(* CoDeSys 2.3 library: TcMc2Drive.lib *)
(* Libraries: STANDARD.LIB 5.6.98 11:03:02, TcBase.lib 14.5.09 11:14:08, TcSystem.lib 10.9.09 11:54:20, TcUtilities.lib 13.10.09 07:46:56, TcEtherCAT.lib 15.1.10 19:43:55, TcTestAndSet.lib 23.2.09 11:50:08, TcDrive.lib 19.1.10 09:32:20, TcBaseMath.lib 27.7.04 11:07:56, TcMath.lib 23.9.04 14:15:30, TcMC2.lib 18.11.09 13:36:54 *)

(* POU F_GetVersionTcMc2Drive, ST *)
FUNCTION F_GetVersionTcMc2Drive : UINT
(* Returns the library version information  *)
VAR_INPUT
	nVersionElement       :       INT;
END_VAR
VAR
END_VAR
(* Version history:
Date          		| Version 		| created under 	     	| Author    | Remark 
------------------------------------------------------------------------------------------------------------------------------------------------------ 
15.05.2008    		| 0.0.1      	| V2.10.0 (Build 1325) 		| I.Ch.		| first release 
13.06.2008    		| 0.0.2      	| V2.10.0 (Build 1325) 		| I.Ch.		| FB_SoEAX5000Reset added  
10.07.2008    		| 0.0.3      	| V2.10.0 (Build 1326) 		| PKa		| FB_SoEAX5000Reset interface update/bugfix  
11.07.2008    		| 0.0.4      	| V2.10.0 (Build 1328) 		| PKa		| FB_SoEAX5000Reset AdsWrite call with falling edge, NC reset timer set to 1sec 
28.07.2008    		| 0.0.5      	| V2.10.0 (Build 1328) 		| I.Ch.		| using ST_DriveRef instead of ST_SoE_DriveRef
18.08.2008    		| 0.0.6      	| V2.10.0 (Build 1328) 		| I.Ch.		| Axis as VAR_IN_OUT
29.08.2008    		| 0.0.7      	| V2.10.0 (Build 1328) 		| I.Ch.		| FB_SoEAX5000Reset removed, FB_SoEReset modified
24.09.2008			| 0.0.8			| V2.10.0 (Build 1328)		| AnK		| FB_SoEReset: internal NC reset removed
02.10.2008			| 0.0.9			| V2.10.0 (Build 1328)		| I.Ch.		| folders added
03.10.2008			| 0.0.10		| V2.10.0 (Build 1330)		| I.Ch.		| created from TcNcDrive.lib v0.0.9
12.12.2008			| 0.0.11		| V2.10.0 (Build 1330)		| I.Ch.		| FB_SoEAX5000FirmwareUpdate added
15.12.2008			| 0.0.13		| V2.10.0 (Build 1330)		| I.Ch.		| cleanup
16.12.2008			| 0.0.14		| V2.10.0 (Build 1330)		| I.Ch.		| provide FB_EcFoeLoad.sInfo as iDiagNumber
16.01.2009			| 0.0.15		| V2.10.0 (Build 1331)		| I.Ch.		| update library list
05.02.2009			| 0.0.19		| V2.10.0 (Build 1332)		| I.Ch.		| cleanup
15.03.2009			| 0.0.20		| V2.11.0 (Build 1534)		| I.Ch.		| FB_SoEReadClassXDiag added, reads C1D|C2D|C3D class diag 
23.03.2009			| 0.0.22		| V2.11.0 (Build 1539)		| I.Ch.		| update library manager
13.01.2010			| 0.0.25		| V2.11.0 (Build 1541)		| I.Ch.		| flexible length for diagnumber list in FB_SoEReadDiagNumberList 
*)
CASE nVersionElement OF
1: (* major number *)
       F_GetVersionTcMc2Drive := 0;
2: (* minor number *)
       F_GetVersionTcMc2Drive := 0;
3: (* revision number *)
       F_GetVersionTcMc2Drive := 25;
ELSE
   F_GetVersionTcMc2Drive := 16#FFFF;
END_CASE
END_FUNCTION

(* POU FB_SoEAX5000FirmwareUpdate, ST *)
FUNCTION_BLOCK FB_SoEAX5000FirmwareUpdate
VAR_INPUT
	sNetId					: T_AmsNetId := '';	(* netID of PC with NC *)
	bExecute				: BOOL;				(* Function block execution is triggered by a rising edge at this input.*)
	sFirmwareVersion		: STRING(20);		(* version string vx_yy_bnnnn, e.g. "v1.05_b0009" for v1.05 Build 0009*)
	sFirmwarePath			: T_MaxString;		(* drive:\path, e.g. "C:\TwinCAT\Io\TcDriveManager\FirmwarePool" *)
	iReqEcState				: UINT := EC_DEVICE_STATE_OP;
	tTimeout				: TIME := DEFAULT_ADS_TIMEOUT;(* States the time before the function is cancelled. *)
END_VAR
VAR_IN_OUT
	Axis					: AXIS_REF;	(* Axis reference *)
END_VAR
VAR_OUTPUT
	bBusy					: BOOL;
	bError					: BOOL;
	iAdsErrId				: UINT;
	iSercosErrId			: UINT;
	iDiagNumber				: UDINT;
	eFwUpdateState			: E_FwUpdateState;
	iLoadProgress			: INT;
	sSelectedFirmwareFile	: STRING(MAX_STRING_LENGTH);	(* found firmware file, e.g. "AX5yxx_xxxx_0010_v1_05_b0009.efw" *)
END_VAR
{library private}
VAR
	fbSoEFirmwareUpdate		: FB_SoEAX5000FirmwareUpdate_ByDriveRef;
	iState					: INT;
	bExecute_I				: BOOL;
   	nAxisId_I      			: DWORD;
	fbAdsRead				: ADSREAD;
	readBuffer				: ARRAY[0..9] OF BYTE;
	nIds					: T_AmsNetIdArr; (* Ams net id as array of bytes *)
	stDriveRef				: ST_DriveRef; (* contains sNetID of EcMaster, nSlaveAddr of EcDrive, nDriveNo of EcDrive, either preset or read from NC *)
END_VAR
VAR CONSTANT
	NCIDXG_AXPARMS			: UDINT := 16#00004000;	(* Axis with ID: Parameter 			*)
	NCIDXO_AXP_HWAMSADDR	: UDINT := 16#00000031;
END_VAR
CASE iState OF
0: (* idle *)
	IF bExecute AND NOT bExecute_I THEN
		bExecute_I := bExecute;

		(* use axis id to determine stDriveRef *)
		IF (Axis.NcToPlc.AxisId = nAxisId_I) AND (stDriveRef.nSlaveAddr <> 0)  AND (stDriveRef.sNetId <> '') THEN
			(* Axis ID unchanged, reference available *)
			iState := 20; (* use reference *)
		ELSE
			(* Axis ID changed *)
			iState := 10; (* get reference from NC *)
			MEMSET(ADR(stDriveRef), 0, SIZEOF(stDriveRef));
			MEMSET(ADR(readBuffer), 0, SIZEOF(readBuffer));

			fbAdsRead(
				NETID	:= sNetId,
				PORT	:= AMSPORT_R0_NC,
				IDXGRP	:= NCIDXG_AXPARMS + Axis.NcToPlc.AxisId,
				IDXOFFS	:= NCIDXO_AXP_HWAMSADDR,
				LEN		:= SIZEOF(readBuffer) ,
				DESTADDR:= ADR(readBuffer),
				READ	:= FALSE,
				TMOUT	:= tTimeout
			);
			fbAdsRead(READ := TRUE);

		END_IF

		nAxisId_I 	:= Axis.NcToPlc.AxisId;
		bBusy		:= TRUE;
		bError		:= FALSE;
		iAdsErrId		:= 0;
		iSercosErrId	:= 0;
		iDiagNumber		:= 0;
		eFwUpdateState			:= eFwU_NoError;
		iLoadProgress			:= 0;
		sSelectedFirmwareFile	:= '';
	END_IF

10: (* get reference from NC *)
	fbAdsRead(READ := FALSE);
	IF NOT fbAdsRead.BUSY THEN
		fbAdsRead(READ := FALSE);

		IF NOT fbAdsRead.ERR THEN
			MEMCPY(ADR(nIds), ADR(readBuffer), SIZEOF(nIds)); 										(* readBuffer[0..5] *)
			MEMCPY(ADR(stDriveRef.nSlaveAddr), ADR(readBuffer[6]), SIZEOF(stDriveRef.nSlaveAddr));  	(* readBuffer[6..7] *)
			MEMCPY(ADR(stDriveRef.nDriveNo), ADR(readBuffer[8]), SIZEOF(stDriveRef.nDriveNo));  		(* readBuffer[8..9] *)

			(* create string out of byte array *)
			stDriveRef.sNetId := F_CreateAmsNetId(nIds);
			iState	:= 20;
		ELSE
			bBusy	:= FALSE;
			bError	:= TRUE;
			iAdsErrId	:= UDINT_TO_UINT(fbAdsRead.ERRID);
			iState	:= 0;
		END_IF
	END_IF

20: (* check and update firmware *)
	fbSoEFirmwareUpdate(
		stDriveRef		:= stDriveRef,
		bExecute		:= FALSE,
		sFirmwareVersion:= sFirmwareVersion,
		sFirmwarePath	:= sFirmwarePath,
		sNetIdIPC		:= sNetId,
		iReqEcState		:= iReqEcState,
		tTimeout		:= tTimeout
	);

	fbSoEFirmwareUpdate(bExecute := TRUE);
	iState	:= 30;

30: (* wait for check and update firmware done *)
	fbSoEFirmwareUpdate(
		bExecute 				:= FALSE,
		eFwUpdateState 			=> eFwUpdateState,
		iLoadProgress			=> iLoadProgress,
		sSelectedFirmwareFile 	=> sSelectedFirmwareFile,
	);

	IF NOT fbSoEFirmwareUpdate.bBusy THEN
		fbSoEFirmwareUpdate(
			bExecute 				:= FALSE,
			eFwUpdateState 			=> eFwUpdateState,
			iLoadProgress			=> iLoadProgress,
			sSelectedFirmwareFile 	=> sSelectedFirmwareFile,
		);
		iState	:= 0;

		IF NOT fbSoEFirmwareUpdate.bError THEN
			bBusy	:= FALSE;
		ELSE
			bBusy	:= FALSE;
			bError	:= TRUE;
			iAdsErrId		:= fbSoEFirmwareUpdate.iAdsErrId;
			iSercosErrId	:= fbSoEFirmwareUpdate.iSercosErrId;
			iDiagNumber		:= fbSoEFirmwareUpdate.iDiagNumber;
		END_IF
	END_IF

END_CASE

bExecute_I := bExecute_I AND bExecute;
END_FUNCTION_BLOCK

(* POU FB_SoEAX5000ReadActMainVoltage, ST *)
FUNCTION_BLOCK FB_SoEAX5000ReadActMainVoltage
VAR_INPUT
	NetId					: T_AmsNetId := '';	(* netID of PC with NC *)
	Execute					: BOOL;				(* Function block execution is triggered by a rising edge at this input.*)
	Timeout					: TIME := DEFAULT_ADS_TIMEOUT;(* States the time before the function is cancelled. *)
END_VAR
VAR_IN_OUT
	Axis					: AXIS_REF;	(* Axis reference *)
END_VAR
VAR_OUTPUT
	Busy					: BOOL;
	Error					: BOOL;
	AdsErrId				: UINT;
	SercosErrId				: UINT;
	Attribute				: DWORD;
	ActualMainVoltage		: LREAL;
END_VAR
{library private}
VAR
	fbEcSoEReadActMainVolt	: FB_SoEAX5000ReadActMainVoltage_ByDriveRef;
	iState					: INT;
	bExecute_I				: BOOL;
   	nAxisId_I      			: DWORD;
	fbAdsRead				: ADSREAD;
	readBuffer				: ARRAY[0..9] OF BYTE;
	nIds					: T_AmsNetIdArr; (* Ams net id as array of bytes *)
	stDriveRef				: ST_DriveRef; (* contains sNetID of EcMaster, nSlaveAddr of EcDrive, nDriveNo of EcDrive, either preset or read from NC *)
END_VAR
VAR CONSTANT
	NCIDXG_AXPARMS			: UDINT := 16#00004000;	(* Axis with ID: Parameter 			*)
	NCIDXO_AXP_HWAMSADDR	: UDINT := 16#00000031;
END_VAR
CASE iState OF
0: (* idle *)
	IF Execute AND NOT bExecute_I THEN
		bExecute_I := Execute;

		(* use axis id to determine stDriveRef *)
		IF (Axis.NcToPlc.AxisId = nAxisId_I) AND (stDriveRef.nSlaveAddr <> 0)  AND (stDriveRef.sNetId <> '') THEN
			(* Axis ID unchanged, reference available *)
			iState := 20; (* use reference *)
		ELSE
			(* Axis ID changed *)
			iState := 10; (* get reference from NC *)
			MEMSET(ADR(stDriveRef), 0, SIZEOF(stDriveRef));
			MEMSET(ADR(readBuffer), 0, SIZEOF(readBuffer));

			fbAdsRead(
				NETID	:= NetId,
				PORT	:= AMSPORT_R0_NC,
				IDXGRP	:= NCIDXG_AXPARMS + Axis.NcToPlc.AxisId,
				IDXOFFS	:= NCIDXO_AXP_HWAMSADDR,
				LEN		:= SIZEOF(readBuffer) ,
				DESTADDR:= ADR(readBuffer),
				READ	:= FALSE,
				TMOUT	:= Timeout
			);
			fbAdsRead(READ := TRUE);

		END_IF

		nAxisId_I 	:= Axis.NcToPlc.AxisId;
		Busy		:= TRUE;
		Error		:= FALSE;
		AdsErrId	:= 0;
		SercosErrId	:= 0;
	END_IF

10: (* get reference from NC *)
	fbAdsRead(READ := FALSE);
	IF NOT fbAdsRead.BUSY THEN
		fbAdsRead(READ := FALSE);

		IF NOT fbAdsRead.ERR THEN
			MEMCPY(ADR(nIds), ADR(readBuffer), SIZEOF(nIds)); 										(* readBuffer[0..5] *)
			MEMCPY(ADR(stDriveRef.nSlaveAddr), ADR(readBuffer[6]), SIZEOF(stDriveRef.nSlaveAddr));  	(* readBuffer[6..7] *)
			MEMCPY(ADR(stDriveRef.nDriveNo), ADR(readBuffer[8]), SIZEOF(stDriveRef.nDriveNo));  		(* readBuffer[8..9] *)

			(* create string out of byte array *)
			stDriveRef.sNetId := F_CreateAmsNetId(nIds);
			iState	:= 20;
		ELSE
			Busy	:= FALSE;
			Error	:= TRUE;
			AdsErrId	:= UDINT_TO_UINT(fbAdsRead.ERRID);
			iState	:= 0;
			Attribute := 0;
			ActualMainVoltage := 0;
		END_IF
	END_IF

20: (* read actual main voltage *)
	fbEcSoEReadActMainVolt(
		stDriveRef		:= stDriveRef,
		bExecute		:= FALSE,
		tTimeout		:= Timeout
	);
	fbEcSoEReadActMainVolt(bExecute := TRUE);
	iState	:= 30;

30: (* wait for read actual main voltage done *)
	fbEcSoEReadActMainVolt(bExecute := FALSE);

	IF NOT fbEcSoEReadActMainVolt.bBusy THEN
		fbEcSoEReadActMainVolt(bExecute := FALSE);
		iState	:= 0;

		IF NOT fbEcSoEReadActMainVolt.bError THEN
			Busy	:= FALSE;
			ActualMainVoltage 	:= fbEcSoEReadActMainVolt.fActualMainVoltage;
			Attribute 			:=  fbEcSoEReadActMainVolt.dwAttribute;
		ELSE
			Busy	:= FALSE;
			Error	:= TRUE;
			AdsErrId		:= fbEcSoEReadActMainVolt.iAdsErrId;
			SercosErrId		:= fbEcSoEReadActMainVolt.iSercosErrId;
			Attribute 		:=  fbEcSoEReadActMainVolt.dwAttribute;
			ActualMainVoltage := 0;
		END_IF
	END_IF

END_CASE

bExecute_I := bExecute_I AND Execute;
END_FUNCTION_BLOCK

(* POU FB_SoEAX5000SetMotorCtrlWord, ST *)
FUNCTION_BLOCK FB_SoEAX5000SetMotorCtrlWord
VAR_INPUT
	NetId			: T_AmsNetId := '';	(* netID of PC with NC *)
	Execute			: BOOL;				(* Function block execution is triggered by a rising edge at this input.*)
	Timeout			: TIME := DEFAULT_ADS_TIMEOUT;(* States the time before the function is cancelled. *)
	ForceLock		: BOOL;
	ForceUnlock		: BOOL;
END_VAR
VAR_IN_OUT
	Axis			: AXIS_REF;	(* Axis reference *)
END_VAR
VAR_OUTPUT
	Busy			: BOOL;
	Error			: BOOL;
	AdsErrId		: UINT;
	SercosErrId		: UINT;
END_VAR
{library private}
VAR
	fbEcSoESetMotorCtrlWord	: FB_SoEAX5000SetMotorCtrlWord_ByDriveRef;
	iState			: INT;
	bExecute_I		: BOOL;
   	nAxisId_I      	: DWORD;
	fbAdsRead		: ADSREAD;
	readBuffer		: ARRAY[0..9] OF BYTE;
	nIds			: T_AmsNetIdArr; (* Ams net id as array of bytes *)
	stDriveRef		: ST_DriveRef; (* contains sNetID of EcMaster, nSlaveAddr of EcDrive, nDriveNo of EcDrive, either preset or read from NC *)
END_VAR
VAR CONSTANT
	NCIDXG_AXPARMS			: UDINT := 16#00004000;	(* Axis with ID: Parameter 			*)
	NCIDXO_AXP_HWAMSADDR	: UDINT := 16#00000031;
END_VAR
CASE iState OF
0: (* idle *)
	IF Execute AND NOT bExecute_I THEN
		bExecute_I := Execute;

		(* use axis id to determine stDriveRef *)
		IF (Axis.NcToPlc.AxisId = nAxisId_I) AND (stDriveRef.nSlaveAddr <> 0)  AND (stDriveRef.sNetId <> '') THEN
			(* Axis ID unchanged, reference available *)
			iState := 20; (* use reference *)
		ELSE
			(* Axis ID changed *)
			iState := 10; (* get reference from NC *)
			MEMSET(ADR(stDriveRef), 0, SIZEOF(stDriveRef));
			MEMSET(ADR(readBuffer), 0, SIZEOF(readBuffer));

			fbAdsRead(
				NETID	:= NetId,
				PORT	:= AMSPORT_R0_NC,
				IDXGRP	:= NCIDXG_AXPARMS + Axis.NcToPlc.AxisId,
				IDXOFFS	:= NCIDXO_AXP_HWAMSADDR,
				LEN		:= SIZEOF(readBuffer) ,
				DESTADDR:= ADR(readBuffer),
				READ	:= FALSE,
				TMOUT	:= Timeout
			);
			fbAdsRead(READ := TRUE);

		END_IF

		nAxisId_I 	:= Axis.NcToPlc.AxisId;
		Busy		:= TRUE;
		Error		:= FALSE;
		AdsErrId		:= 0;
		SercosErrId	:= 0;
	END_IF

10: (* get reference from NC *)
	fbAdsRead(READ := FALSE);
	IF NOT fbAdsRead.BUSY THEN
		fbAdsRead(READ := FALSE);

		IF NOT fbAdsRead.ERR THEN
			MEMCPY(ADR(nIds), ADR(readBuffer), SIZEOF(nIds)); 										(* readBuffer[0..5] *)
			MEMCPY(ADR(stDriveRef.nSlaveAddr), ADR(readBuffer[6]), SIZEOF(stDriveRef.nSlaveAddr));  	(* readBuffer[6..7] *)
			MEMCPY(ADR(stDriveRef.nDriveNo), ADR(readBuffer[8]), SIZEOF(stDriveRef.nDriveNo));  		(* readBuffer[8..9] *)

			(* create string out of byte array *)
			stDriveRef.sNetId := F_CreateAmsNetId(nIds);
			iState	:= 20;
		ELSE
			Busy	:= FALSE;
			Error	:= TRUE;
			AdsErrId:= UDINT_TO_UINT(fbAdsRead.ERRID);
			iState	:= 0;
		END_IF
	END_IF

20: (* set motor control word *)
	fbEcSoESetMotorCtrlWord(
		stDriveRef		:= stDriveRef,
		bExecute		:= FALSE,
		tTimeout		:= Timeout,
		bForceLock		:= ForceLock,
		bForceUnlock	:= ForceUnlock
	);
	fbEcSoESetMotorCtrlWord(bExecute := TRUE);
	iState	:= 30;

30: (* wait for set motor control word done *)
	fbEcSoESetMotorCtrlWord(bExecute := FALSE);

	IF NOT fbEcSoESetMotorCtrlWord.bBusy THEN
		fbEcSoESetMotorCtrlWord(bExecute := FALSE);
		iState	:= 0;

		IF NOT fbEcSoESetMotorCtrlWord.bError THEN
			Busy	:= FALSE;
		ELSE
			Busy	:= FALSE;
			Error	:= TRUE;
			AdsErrId	:= fbEcSoESetMotorCtrlWord.iAdsErrId;
			SercosErrId	:= fbEcSoESetMotorCtrlWord.iSercosErrId;
		END_IF
	END_IF

END_CASE

bExecute_I := bExecute_I AND Execute;
END_FUNCTION_BLOCK

(* POU FB_SoEExecuteCommand, ST *)
FUNCTION_BLOCK FB_SoEExecuteCommand
VAR_INPUT
	NetId			: T_AmsNetId := '';	(* netID of PC with NC *)
	Idn				: WORD;				(* SoE IDN: e.g. "S_0_IDN + 1" for S-0-0001 or "P_0_IDN + 23" for P-0-0023*)
	Execute			: BOOL;				(* Function block execution is triggered by a rising edge at this input.*)
	Timeout			: TIME := DEFAULT_ADS_TIMEOUT;(* States the time before the function is cancelled. *)
END_VAR
VAR_IN_OUT
	Axis			: AXIS_REF;	(* Axis reference *)
END_VAR
VAR_OUTPUT
	Busy			: BOOL;
	Error			: BOOL;
	AdsErrId		: UINT;
	SercosErrId		: UINT;
END_VAR
{library private}
VAR
	fbEcSoECommand	: FB_SoEExecuteCommand_ByDriveRef;
	iState			: INT;
	bExecute_I		: BOOL;
   	nAxisId_I      	: DWORD;
	fbAdsRead		: ADSREAD;
	readBuffer		: ARRAY[0..9] OF BYTE;
	nIds			: T_AmsNetIdArr; (* Ams net id as array of bytes *)
	stDriveRef		: ST_DriveRef; (* contains sNetID of EcMaster, nSlaveAddr of EcDrive, nDriveNo of EcDrive, either preset or read from NC *)
END_VAR
VAR CONSTANT
	NCIDXG_AXPARMS			: UDINT := 16#00004000;	(* Axis with ID: Parameter 			*)
	NCIDXO_AXP_HWAMSADDR	: UDINT := 16#00000031;
END_VAR
CASE iState OF
0: (* idle *)
	IF Execute AND NOT bExecute_I THEN
		bExecute_I := Execute;

		(* use axis id to determine stDriveRef *)
		IF (Axis.NcToPlc.AxisId = nAxisId_I) AND (stDriveRef.nSlaveAddr <> 0)  AND (stDriveRef.sNetId <> '') THEN
			(* Axis ID unchanged, reference available *)
			iState := 20; (* use reference *)
		ELSE
			(* Axis ID changed *)
			iState := 10; (* get reference from NC *)
			MEMSET(ADR(stDriveRef), 0, SIZEOF(stDriveRef));
			MEMSET(ADR(readBuffer), 0, SIZEOF(readBuffer));

			fbAdsRead(
				NETID	:= NetId,
				PORT	:= AMSPORT_R0_NC,
				IDXGRP	:= NCIDXG_AXPARMS + Axis.NcToPlc.AxisId,
				IDXOFFS	:= NCIDXO_AXP_HWAMSADDR,
				LEN		:= SIZEOF(readBuffer) ,
				DESTADDR:= ADR(readBuffer),
				READ	:= FALSE,
				TMOUT	:= Timeout
			);
			fbAdsRead(READ := TRUE);

		END_IF

		nAxisId_I 	:= Axis.NcToPlc.AxisId;
		Busy		:= TRUE;
		Error		:= FALSE;
		AdsErrId	:= 0;
		SercosErrId	:= 0;
	END_IF

10: (* get reference from NC *)
	fbAdsRead(READ := FALSE);
	IF NOT fbAdsRead.BUSY THEN
		fbAdsRead(READ := FALSE);

		IF NOT fbAdsRead.ERR THEN
			MEMCPY(ADR(nIds), ADR(readBuffer), SIZEOF(nIds)); 										(* readBuffer[0..5] *)
			MEMCPY(ADR(stDriveRef.nSlaveAddr), ADR(readBuffer[6]), SIZEOF(stDriveRef.nSlaveAddr));  	(* readBuffer[6..7] *)
			MEMCPY(ADR(stDriveRef.nDriveNo), ADR(readBuffer[8]), SIZEOF(stDriveRef.nDriveNo));  		(* readBuffer[8..9] *)

			(* create string out of byte array *)
			stDriveRef.sNetId := F_CreateAmsNetId(nIds);
			iState	:= 20;
		ELSE
			Busy	:= FALSE;
			Error	:= TRUE;
			AdsErrId:= UDINT_TO_UINT(fbAdsRead.ERRID);
			iState	:= 0;
		END_IF
	END_IF

20: (* write SoE command *)
	fbEcSoECommand(
		stDriveRef		:= stDriveRef,
		nIdn			:= Idn,
		bExecute		:= FALSE,
		tTimeout		:= Timeout
	);
	fbEcSoECommand(bExecute := TRUE);
	iState	:= 30;

30: (* wait for write SoE data done *)
	fbEcSoECommand(bExecute := FALSE);

	IF NOT fbEcSoECommand.bBusy THEN
		fbEcSoECommand(bExecute := FALSE);
		iState	:= 0;

		IF NOT fbEcSoECommand.bError THEN
			Busy	:= FALSE;
		ELSE
			Busy	:= FALSE;
			Error	:= TRUE;
			AdsErrId	:= fbEcSoECommand.iAdsErrId;
			SercosErrId	:= fbEcSoECommand.iSercosErrId;
		END_IF
	END_IF

END_CASE

bExecute_I := bExecute_I AND Execute;
END_FUNCTION_BLOCK

(* POU FB_SoERead, ST *)
FUNCTION_BLOCK FB_SoERead
VAR_INPUT
	NetId			: T_AmsNetId := '';	(* netID of PC with NC *)
	Idn				: WORD;				(* SoE IDN: e.g. "S_0_IDN + 1" for S-0-0001 or "P_0_IDN + 23" for P-0-0023*)
	Element			: BYTE;				(* SoE element.*)
	pDstBuf			: DWORD;			(* Contains the address of the buffer for the received data. *)
	BufLen			: UDINT;			(* Contains the max. number of bytes to be received. *)
	Execute			: BOOL;				(* Function block execution is triggered by a rising edge at this input.*)
	Timeout			: TIME := DEFAULT_ADS_TIMEOUT;(* States the time before the function is cancelled. *)
END_VAR
VAR_IN_OUT
	Axis			: AXIS_REF;	(* Axis reference *)
END_VAR
VAR_OUTPUT
	Busy			: BOOL;
	Error			: BOOL;
	AdsErrId		: UINT;
	SercosErrId		: UINT;
	Attribute		: DWORD;
END_VAR
{library private}
VAR
	fbEcSoEReadEx	: FB_SoERead_ByDriveRef;
	iState			: INT;
	bExecute_I		: BOOL;
   	nAxisId_I      	: DWORD;
	fbAdsRead		: ADSREAD;
	readBuffer		: ARRAY[0..9] OF BYTE;
	nIds			: T_AmsNetIdArr; (* Ams net id as array of bytes *)
	stDriveRef		: ST_DriveRef; (* contains sNetID of EcMaster, nSlaveAddr of EcDrive, nDriveNo of EcDrive, either preset or read from NC *)
END_VAR
VAR CONSTANT
	NCIDXG_AXPARMS			: UDINT := 16#00004000;	(* Axis with ID: Parameter 			*)
	NCIDXO_AXP_HWAMSADDR	: UDINT := 16#00000031;
END_VAR
CASE iState OF
0: (* idle *)
	IF Execute AND NOT bExecute_I THEN
		bExecute_I := Execute;

		(* use axis id to determine stDriveRef *)
		IF (Axis.NcToPlc.AxisId = nAxisId_I) AND (stDriveRef.nSlaveAddr <> 0)  AND (stDriveRef.sNetId <> '') THEN
			(* Axis ID unchanged, reference available *)
			iState := 20; (* use reference *)
		ELSE
			(* Axis ID changed *)
			iState := 10; (* get reference from NC *)
			MEMSET(ADR(stDriveRef), 0, SIZEOF(stDriveRef));
			MEMSET(ADR(readBuffer), 0, SIZEOF(readBuffer));

			fbAdsRead(
				NETID	:= NetId,
				PORT	:= AMSPORT_R0_NC,
				IDXGRP	:= NCIDXG_AXPARMS + Axis.NcToPlc.AxisId,
				IDXOFFS	:= NCIDXO_AXP_HWAMSADDR,
				LEN		:= SIZEOF(readBuffer) ,
				DESTADDR:= ADR(readBuffer),
				READ	:= FALSE,
				TMOUT	:= Timeout
			);
			fbAdsRead(READ := TRUE);

		END_IF

		nAxisId_I 	:= Axis.NcToPlc.AxisId;
		Busy		:= TRUE;
		Error		:= FALSE;
		AdsErrId	:= 0;
		SercosErrId	:= 0;
	END_IF

10: (* get reference from NC *)
	fbAdsRead(READ := FALSE);
	IF NOT fbAdsRead.BUSY THEN
		fbAdsRead(READ := FALSE);

		IF NOT fbAdsRead.ERR THEN
			MEMCPY(ADR(nIds), ADR(readBuffer), SIZEOF(nIds)); 										(* readBuffer[0..5] *)
			MEMCPY(ADR(stDriveRef.nSlaveAddr), ADR(readBuffer[6]), SIZEOF(stDriveRef.nSlaveAddr));  	(* readBuffer[6..7] *)
			MEMCPY(ADR(stDriveRef.nDriveNo), ADR(readBuffer[8]), SIZEOF(stDriveRef.nDriveNo));  		(* readBuffer[8..9] *)

			(* create string out of byte array *)
			stDriveRef.sNetId := F_CreateAmsNetId(nIds);
			iState	:= 20;
		ELSE
			Busy	:= FALSE;
			Error	:= TRUE;
			AdsErrId	:= UDINT_TO_UINT(fbAdsRead.ERRID);
			Attribute 	:= 0;
			iState	:= 0;
		END_IF
	END_IF

20: (* read SoE data *)
	fbEcSoEReadEx(
		stDriveRef		:= stDriveRef,
		nIdn			:= Idn,
		nElement		:= Element,
		pDstBuf			:= pDstBuf,
		cbBufLen		:= BufLen,
		bExecute		:= FALSE,
		tTimeout		:= Timeout
	);
	fbEcSoEReadEx(bExecute := TRUE);
	iState	:= 30;

30: (* wait for read SoE data done *)
	fbEcSoEReadEx(bExecute := FALSE);

	IF NOT fbEcSoEReadEx.bBusy THEN
		fbEcSoEReadEx(bExecute := FALSE);
		iState	:= 0;
		Attribute := fbEcSoEReadEx.dwAttribute;

		IF NOT fbEcSoEReadEx.bError THEN
			Busy	:= FALSE;
		ELSE
			Busy	:= FALSE;
			Error	:= TRUE;
			AdsErrId	:= fbEcSoEReadEx.iAdsErrId;
			SercosErrId	:= fbEcSoEReadEx.iSercosErrId;
		END_IF
	END_IF

END_CASE

bExecute_I := bExecute_I AND Execute;
END_FUNCTION_BLOCK

(* POU FB_SoEReadAmplifierTemperature, ST *)
FUNCTION_BLOCK FB_SoEReadAmplifierTemperature
VAR_INPUT
	NetId					: T_AmsNetId := '';	(* netID of PC with NC *)
	Execute					: BOOL;				(* Function block execution is triggered by a rising edge at this input.*)
	Timeout					: TIME := DEFAULT_ADS_TIMEOUT;(* States the time before the function is cancelled. *)
END_VAR
VAR_IN_OUT
	Axis					: AXIS_REF;	(* Axis reference *)
END_VAR
VAR_OUTPUT
	Busy					: BOOL;
	Error					: BOOL;
	AdsErrId				: UINT;
	SercosErrId				: UINT;
	AmplifierTemperature	: REAL;
	Attribute				: DWORD;
END_VAR
{library private}
VAR
	fbEcSoEReadAmplifierTemp: FB_SoEReadAmplifierTemperature_ByDriveRef;
	iState					: INT;
	bExecute_I				: BOOL;
   	nAxisId_I      			: DWORD;
	fbAdsRead				: ADSREAD;
	readBuffer				: ARRAY[0..9] OF BYTE;
	nIds					: T_AmsNetIdArr; (* Ams net id as array of bytes *)
	stDriveRef				: ST_DriveRef; (* contains sNetID of EcMaster, nSlaveAddr of EcDrive, nDriveNo of EcDrive, either preset or read from NC *)
END_VAR
VAR CONSTANT
	NCIDXG_AXPARMS			: UDINT := 16#00004000;	(* Axis with ID: Parameter 			*)
	NCIDXO_AXP_HWAMSADDR	: UDINT := 16#00000031;
END_VAR
CASE iState OF
0: (* idle *)
	IF Execute AND NOT bExecute_I THEN
		bExecute_I := Execute;

		(* use axis id to determine stDriveRef *)
		IF (Axis.NcToPlc.AxisId = nAxisId_I) AND (stDriveRef.nSlaveAddr <> 0)  AND (stDriveRef.sNetId <> '') THEN
			(* Axis ID unchanged, reference available *)
			iState := 20; (* use reference *)
		ELSE
			(* Axis ID changed *)
			iState := 10; (* get reference from NC *)
			MEMSET(ADR(stDriveRef), 0, SIZEOF(stDriveRef));
			MEMSET(ADR(readBuffer), 0, SIZEOF(readBuffer));

			fbAdsRead(
				NETID	:= NetId,
				PORT	:= AMSPORT_R0_NC,
				IDXGRP	:= NCIDXG_AXPARMS + Axis.NcToPlc.AxisId,
				IDXOFFS	:= NCIDXO_AXP_HWAMSADDR,
				LEN		:= SIZEOF(readBuffer) ,
				DESTADDR:= ADR(readBuffer),
				READ	:= FALSE,
				TMOUT	:= Timeout
			);
			fbAdsRead(READ := TRUE);

		END_IF

		nAxisId_I 	:= Axis.NcToPlc.AxisId;
		Busy		:= TRUE;
		Error		:= FALSE;
		AdsErrId	:= 0;
		SercosErrId	:= 0;
	END_IF

10: (* get reference from NC *)
	fbAdsRead(READ := FALSE);
	IF NOT fbAdsRead.BUSY THEN
		fbAdsRead(READ := FALSE);

		IF NOT fbAdsRead.ERR THEN
			MEMCPY(ADR(nIds), ADR(readBuffer), SIZEOF(nIds)); 										(* readBuffer[0..5] *)
			MEMCPY(ADR(stDriveRef.nSlaveAddr), ADR(readBuffer[6]), SIZEOF(stDriveRef.nSlaveAddr));  	(* readBuffer[6..7] *)
			MEMCPY(ADR(stDriveRef.nDriveNo), ADR(readBuffer[8]), SIZEOF(stDriveRef.nDriveNo));  		(* readBuffer[8..9] *)

			(* create string out of byte array *)
			stDriveRef.sNetId := F_CreateAmsNetId(nIds);
			iState	:= 20;
		ELSE
			Busy	:= FALSE;
			Error	:= TRUE;
			AdsErrId	:= UDINT_TO_UINT(fbAdsRead.ERRID);
			iState		:= 0;
			Attribute 	:= 0;
			AmplifierTemperature := 0;
		END_IF
	END_IF

20: (* read Amplifier Temperature *)
	fbEcSoEReadAmplifierTemp(
		stDriveRef		:= stDriveRef,
		bExecute		:= FALSE,
		tTimeout		:= Timeout
	);
	fbEcSoEReadAmplifierTemp(bExecute := TRUE);
	iState	:= 30;

30: (* wait for read Amplifier Temperature done *)
	fbEcSoEReadAmplifierTemp(bExecute := FALSE);

	IF NOT fbEcSoEReadAmplifierTemp.bBusy THEN
		fbEcSoEReadAmplifierTemp(bExecute := FALSE);
		iState	:= 0;

		IF NOT fbEcSoEReadAmplifierTemp.bError THEN
			Busy	:= FALSE;
			AmplifierTemperature := fbEcSoEReadAmplifierTemp.fAmplifierTemperature;
			Attribute 	:=  fbEcSoEReadAmplifierTemp.dwAttribute;
		ELSE
			Busy	:= FALSE;
			Error	:= TRUE;
			AdsErrId	:= fbEcSoEReadAmplifierTemp.iAdsErrId;
			SercosErrId	:= fbEcSoEReadAmplifierTemp.iSercosErrId;
			Attribute 	:=  fbEcSoEReadAmplifierTemp.dwAttribute;
			AmplifierTemperature := 0;
		END_IF
	END_IF

END_CASE

bExecute_I := bExecute_I AND Execute;
END_FUNCTION_BLOCK

(* POU FB_SoEReadClassXDiag, ST *)
FUNCTION_BLOCK FB_SoEReadClassXDiag
VAR_INPUT
	NetId			: T_AmsNetId := '';	(* netID of PC with NC *)
	Execute			: BOOL;				(* Function block execution is triggered by a rising edge at this input.*)
	DiagClass		: USINT:= 1;		(* 1: C1D (S-0-0011) is default, 2: C2D (S-0-0012), 3: C3D (S-0-0013) *)
	Timeout			: TIME := DEFAULT_ADS_TIMEOUT;(* States the time before the function is cancelled. *)
END_VAR
VAR_IN_OUT
	Axis			: AXIS_REF;	(* Axis reference *)
END_VAR
VAR_OUTPUT
	Busy			: BOOL;
	Error			: BOOL;
	AdsErrId		: UINT;
	SercosErrId		: UINT;
	ClassXDiag		: WORD;
	Attribute		: DWORD;
END_VAR
{library private}
VAR
	fbSoEReadCXD	: FB_SoEReadClassXDiag_ByDriveRef;
	iState			: INT;
	bExecute_I		: BOOL;
   	nAxisId_I      	: DWORD;
	fbAdsRead		: ADSREAD;
	readBuffer		: ARRAY[0..9] OF BYTE;
	nIds			: T_AmsNetIdArr; (* Ams net id as array of bytes *)
	stDriveRef		: ST_DriveRef; (* contains sNetID of EcMaster, nSlaveAddr of EcDrive, nDriveNo of EcDrive, either preset or read from NC *)
END_VAR
VAR CONSTANT
	NCIDXG_AXPARMS			: UDINT := 16#00004000;	(* Axis with ID: Parameter 			*)
	NCIDXO_AXP_HWAMSADDR	: UDINT := 16#00000031;
END_VAR
CASE iState OF
0: (* idle *)
	IF Execute AND NOT bExecute_I THEN
		bExecute_I := Execute;

		(* use axis id to determine stDriveRef *)
		IF (Axis.NcToPlc.AxisId = nAxisId_I) AND (stDriveRef.nSlaveAddr <> 0)  AND (stDriveRef.sNetId <> '') THEN
			(* Axis ID unchanged, reference available *)
			iState := 20; (* use reference *)
		ELSE
			(* Axis ID changed *)
			iState := 10; (* get reference from NC *)
			MEMSET(ADR(stDriveRef), 0, SIZEOF(stDriveRef));
			MEMSET(ADR(readBuffer), 0, SIZEOF(readBuffer));

			fbAdsRead(
				NETID	:= NetId,
				PORT	:= AMSPORT_R0_NC,
				IDXGRP	:= NCIDXG_AXPARMS + Axis.NcToPlc.AxisId,
				IDXOFFS	:= NCIDXO_AXP_HWAMSADDR,
				LEN		:= SIZEOF(readBuffer) ,
				DESTADDR:= ADR(readBuffer),
				READ	:= FALSE,
				TMOUT	:= Timeout
			);
			fbAdsRead(READ := TRUE);

		END_IF

		nAxisId_I 	:= Axis.NcToPlc.AxisId;
		Busy		:= TRUE;
		Error		:= FALSE;
		AdsErrId	:= 0;
		SercosErrId	:= 0;
	END_IF

10: (* get reference from NC *)
	fbAdsRead(READ := FALSE);
	IF NOT fbAdsRead.BUSY THEN
		fbAdsRead(READ := FALSE);

		IF NOT fbAdsRead.ERR THEN
			MEMCPY(ADR(nIds), ADR(readBuffer), SIZEOF(nIds)); 										(* readBuffer[0..5] *)
			MEMCPY(ADR(stDriveRef.nSlaveAddr), ADR(readBuffer[6]), SIZEOF(stDriveRef.nSlaveAddr));  	(* readBuffer[6..7] *)
			MEMCPY(ADR(stDriveRef.nDriveNo), ADR(readBuffer[8]), SIZEOF(stDriveRef.nDriveNo));  		(* readBuffer[8..9] *)

			(* create string out of byte array *)
			stDriveRef.sNetId := F_CreateAmsNetId(nIds);
			iState	:= 20;
		ELSE
			Busy	:= FALSE;
			Error	:= TRUE;
			AdsErrId:= UDINT_TO_UINT(fbAdsRead.ERRID);
			iState	:= 0;
			Attribute := 0;
			ClassXDiag := 0;
		END_IF
	END_IF

20: (* read drive class x diag *)
	fbSoEReadCXD(
		stDriveRef		:= stDriveRef,
		bExecute		:= FALSE,
		iDiagClass		:= DiagClass,
		tTimeout		:= Timeout
	);
	fbSoEReadCXD(bExecute := TRUE);
	iState	:= 30;

30: (* wait for read drive class x diag done *)
	fbSoEReadCXD(bExecute := FALSE);

	IF NOT fbSoEReadCXD.bBusy THEN
		fbSoEReadCXD(bExecute := FALSE);
		iState	:= 0;

		IF NOT fbSoEReadCXD.bError THEN
			Busy	:= FALSE;
			ClassXDiag := fbSoEReadCXD.wClassXDiag;
			Attribute := fbSoEReadCXD.dwAttribute;
		ELSE
			Busy	:= FALSE;
			Error	:= TRUE;
			AdsErrId	:= fbSoEReadCXD.iAdsErrId;
			SercosErrId	:= fbSoEReadCXD.iSercosErrId;
			Attribute 	:= fbSoEReadCXD.dwAttribute;
			ClassXDiag	:= 0;
		END_IF
	END_IF

END_CASE

bExecute_I := bExecute_I AND Execute;
END_FUNCTION_BLOCK

(* POU FB_SoEReadCommandState, ST *)
FUNCTION_BLOCK FB_SoEReadCommandState
VAR_INPUT
	NetId			: T_AmsNetId := '';	(* netID of PC with NC *)
	Idn				: WORD;				(* SoE IDN: e.g. "S_0_IDN + 1" for S-0-0001 or "P_0_IDN + 23" for P-0-0023*)
	Execute			: BOOL;				(* Function block execution is triggered by a rising edge at this input.*)
	Timeout			: TIME := DEFAULT_ADS_TIMEOUT;(* States the time before the function is cancelled. *)
END_VAR
VAR_IN_OUT
	Axis			: AXIS_REF;	(* Axis reference *)
END_VAR
VAR_OUTPUT
	Busy			: BOOL;
	Error			: BOOL;
	CmdState		: E_SoE_CmdState;
	AdsErrId		: UINT;
	SercosErrId		: UINT;
END_VAR
{library private}
VAR
	fbEcSoECmdState	: FB_SoEReadCommandState_ByDriveRef;
	iState			: INT;
	bExecute_I		: BOOL;
   	nAxisId_I      	: DWORD;
	fbAdsRead		: ADSREAD;
	readBuffer		: ARRAY[0..9] OF BYTE;
	nIds			: T_AmsNetIdArr; (* Ams net id as array of bytes *)
	stDriveRef		: ST_DriveRef; (* contains sNetID of EcMaster, nSlaveAddr of EcDrive, nDriveNo of EcDrive, either preset or read from NC *)
END_VAR
VAR CONSTANT
	NCIDXG_AXPARMS			: UDINT := 16#00004000;	(* Axis with ID: Parameter 			*)
	NCIDXO_AXP_HWAMSADDR	: UDINT := 16#00000031;
END_VAR
CASE iState OF
0: (* idle *)
	IF Execute AND NOT bExecute_I THEN
		bExecute_I := Execute;

		(* use axis id to determine stDriveRef *)
		IF (Axis.NcToPlc.AxisId = nAxisId_I) AND (stDriveRef.nSlaveAddr <> 0)  AND (stDriveRef.sNetId <> '') THEN
			(* Axis ID unchanged, reference available *)
			iState := 20; (* use reference *)
		ELSE
			(* Axis ID changed *)
			iState := 10; (* get reference from NC *)
			MEMSET(ADR(stDriveRef), 0, SIZEOF(stDriveRef));
			MEMSET(ADR(readBuffer), 0, SIZEOF(readBuffer));

			fbAdsRead(
				NETID	:= NetId,
				PORT	:= AMSPORT_R0_NC,
				IDXGRP	:= NCIDXG_AXPARMS + Axis.NcToPlc.AxisId,
				IDXOFFS	:= NCIDXO_AXP_HWAMSADDR,
				LEN		:= SIZEOF(readBuffer) ,
				DESTADDR:= ADR(readBuffer),
				READ	:= FALSE,
				TMOUT	:= Timeout
			);
			fbAdsRead(READ := TRUE);

		END_IF

		nAxisId_I 	:= Axis.NcToPlc.AxisId;
		Busy		:= TRUE;
		Error		:= FALSE;
		AdsErrId	:= 0;
		SercosErrId	:= 0;
	END_IF

10: (* get reference from NC *)
	fbAdsRead(READ := FALSE);
	IF NOT fbAdsRead.BUSY THEN
		fbAdsRead(READ := FALSE);

		IF NOT fbAdsRead.ERR THEN
			MEMCPY(ADR(nIds), ADR(readBuffer), SIZEOF(nIds)); 										(* readBuffer[0..5] *)
			MEMCPY(ADR(stDriveRef.nSlaveAddr), ADR(readBuffer[6]), SIZEOF(stDriveRef.nSlaveAddr));  	(* readBuffer[6..7] *)
			MEMCPY(ADR(stDriveRef.nDriveNo), ADR(readBuffer[8]), SIZEOF(stDriveRef.nDriveNo));  		(* readBuffer[8..9] *)

			(* create string out of byte array *)
			stDriveRef.sNetId := F_CreateAmsNetId(nIds);
			iState	:= 20;
		ELSE
			Busy	:= FALSE;
			Error	:= TRUE;
			AdsErrId:= UDINT_TO_UINT(fbAdsRead.ERRID);
			iState	:= 0;
		END_IF
	END_IF

20: (* read command state *)
	fbEcSoECmdState(
		stDriveRef		:= stDriveRef,
		nIdn			:= Idn,
		bExecute		:= FALSE,
		tTimeout		:= Timeout
	);
	fbEcSoECmdState(bExecute := TRUE);
	iState	:= 30;

30: (* wait for read command state done *)
	fbEcSoECmdState(bExecute := FALSE);

	IF NOT fbEcSoECmdState.bBusy THEN
		fbEcSoECmdState(bExecute := FALSE);
		iState		:= 0;
		CmdState 	:= fbEcSoECmdState.eCmdState;

		IF NOT fbEcSoECmdState.bError THEN
			Busy	:= FALSE;
		ELSE
			Busy	:= FALSE;
			Error	:= TRUE;
			AdsErrId	:= fbEcSoECmdState.iAdsErrId;
			SercosErrId	:= fbEcSoECmdState.iSercosErrId;
		END_IF
	END_IF

END_CASE

bExecute_I := bExecute_I AND Execute;
END_FUNCTION_BLOCK

(* POU FB_SoEReadDcBusCurrent, ST *)
FUNCTION_BLOCK FB_SoEReadDcBusCurrent
VAR_INPUT
	NetId			: T_AmsNetId := '';	(* netID of PC with NC *)
	Execute			: BOOL;				(* Function block execution is triggered by a rising edge at this input.*)
	Timeout			: TIME := DEFAULT_ADS_TIMEOUT;(* States the time before the function is cancelled. *)
END_VAR
VAR_IN_OUT
	Axis			: AXIS_REF;	(* Axis reference *)
END_VAR
VAR_OUTPUT
	Busy			: BOOL;
	Error			: BOOL;
	AdsErrId		: UINT;
	SercosErrId		: UINT;
	DcBusCurrent	: REAL;
	Attribute		: DWORD;
END_VAR
{library private}
VAR
	fbEcSoEReadDcBusCurr	: FB_SoEReadDcBusCurrent_ByDriveRef;
	iState					: INT;
	bExecute_I				: BOOL;
   	nAxisId_I      			: DWORD;
	fbAdsRead				: ADSREAD;
	readBuffer				: ARRAY[0..9] OF BYTE;
	nIds					: T_AmsNetIdArr; (* Ams net id as array of bytes *)
	stDriveRef				: ST_DriveRef; (* contains sNetID of EcMaster, nSlaveAddr of EcDrive, nDriveNo of EcDrive, either preset or read from NC *)
END_VAR
VAR CONSTANT
	NCIDXG_AXPARMS			: UDINT := 16#00004000;	(* Axis with ID: Parameter 			*)
	NCIDXO_AXP_HWAMSADDR	: UDINT := 16#00000031;
END_VAR
CASE iState OF
0: (* idle *)
	IF Execute AND NOT bExecute_I THEN
		bExecute_I := Execute;

		(* use axis id to determine stDriveRef *)
		IF (Axis.NcToPlc.AxisId = nAxisId_I) AND (stDriveRef.nSlaveAddr <> 0)  AND (stDriveRef.sNetId <> '') THEN
			(* Axis ID unchanged, reference available *)
			iState := 20; (* use reference *)
		ELSE
			(* Axis ID changed *)
			iState := 10; (* get reference from NC *)
			MEMSET(ADR(stDriveRef), 0, SIZEOF(stDriveRef));
			MEMSET(ADR(readBuffer), 0, SIZEOF(readBuffer));

			fbAdsRead(
				NETID	:= NetId,
				PORT	:= AMSPORT_R0_NC,
				IDXGRP	:= NCIDXG_AXPARMS + Axis.NcToPlc.AxisId,
				IDXOFFS	:= NCIDXO_AXP_HWAMSADDR,
				LEN		:= SIZEOF(readBuffer) ,
				DESTADDR:= ADR(readBuffer),
				READ	:= FALSE,
				TMOUT	:= Timeout
			);
			fbAdsRead(READ := TRUE);

		END_IF

		nAxisId_I 	:= Axis.NcToPlc.AxisId;
		Busy		:= TRUE;
		Error		:= FALSE;
		AdsErrId	:= 0;
		SercosErrId	:= 0;
	END_IF

10: (* get reference from NC *)
	fbAdsRead(READ := FALSE);
	IF NOT fbAdsRead.BUSY THEN
		fbAdsRead(READ := FALSE);

		IF NOT fbAdsRead.ERR THEN
			MEMCPY(ADR(nIds), ADR(readBuffer), SIZEOF(nIds)); 										(* readBuffer[0..5] *)
			MEMCPY(ADR(stDriveRef.nSlaveAddr), ADR(readBuffer[6]), SIZEOF(stDriveRef.nSlaveAddr));  	(* readBuffer[6..7] *)
			MEMCPY(ADR(stDriveRef.nDriveNo), ADR(readBuffer[8]), SIZEOF(stDriveRef.nDriveNo));  		(* readBuffer[8..9] *)

			(* create string out of byte array *)
			stDriveRef.sNetId := F_CreateAmsNetId(nIds);
			iState	:= 20;
		ELSE
			Busy	:= FALSE;
			Error	:= TRUE;
			AdsErrId	:= UDINT_TO_UINT(fbAdsRead.ERRID);
			iState	:= 0;
			Attribute := 0;
			DcBusCurrent := 0;
		END_IF
	END_IF

20: (* read DC bus current *)
	fbEcSoEReadDcBusCurr(
		stDriveRef		:= stDriveRef,
		bExecute		:= FALSE,
		tTimeout		:= Timeout
	);
	fbEcSoEReadDcBusCurr(bExecute := TRUE);
	iState	:= 30;

30: (* wait for read DC bus current done *)
	fbEcSoEReadDcBusCurr(bExecute := FALSE);

	IF NOT fbEcSoEReadDcBusCurr.bBusy THEN
		fbEcSoEReadDcBusCurr(bExecute := FALSE);
		iState	:= 0;

		IF NOT fbEcSoEReadDcBusCurr.bError THEN
			Busy	:= FALSE;
			DcBusCurrent := fbEcSoEReadDcBusCurr.fDcBusCurrent;
			Attribute   := fbEcSoEReadDcBusCurr.dwAttribute;
		ELSE
			Busy	:= FALSE;
			Error	:= TRUE;
			AdsErrId		:= fbEcSoEReadDcBusCurr.iAdsErrId;
			SercosErrId	:= fbEcSoEReadDcBusCurr.iSercosErrId;
			Attribute 	:= fbEcSoEReadDcBusCurr.dwAttribute;
			DcBusCurrent := 0;
		END_IF
	END_IF

END_CASE

bExecute_I := bExecute_I AND Execute;
END_FUNCTION_BLOCK

(* POU FB_SoEReadDcBusVoltage, ST *)
FUNCTION_BLOCK FB_SoEReadDcBusVoltage
VAR_INPUT
	NetId			: T_AmsNetId := '';	(* netID of PC with NC *)
	Execute			: BOOL;				(* Function block execution is triggered by a rising edge at this input.*)
	Timeout			: TIME := DEFAULT_ADS_TIMEOUT;(* States the time before the function is cancelled. *)
END_VAR
VAR_IN_OUT
	Axis			: AXIS_REF;	(* Axis reference *)
END_VAR
VAR_OUTPUT
	Busy			: BOOL;
	Error			: BOOL;
	AdsErrId		: UINT;
	SercosErrId		: UINT;
	DcBusVoltage	: REAL;
	Attribute		: DWORD;
END_VAR
{library private}
VAR
	fbEcSoEReadDcBusVolt	: FB_SoEReadDcBusVoltage_ByDriveRef;
	iState					: INT;
	bExecute_I				: BOOL;
   	nAxisId_I      			: DWORD;
	fbAdsRead				: ADSREAD;
	readBuffer				: ARRAY[0..9] OF BYTE;
	nIds					: T_AmsNetIdArr; (* Ams net id as array of bytes *)
	stDriveRef				: ST_DriveRef; (* contains sNetID of EcMaster, nSlaveAddr of EcDrive, nDriveNo of EcDrive, either preset or read from NC *)
END_VAR
VAR CONSTANT
	NCIDXG_AXPARMS			: UDINT := 16#00004000;	(* Axis with ID: Parameter 			*)
	NCIDXO_AXP_HWAMSADDR	: UDINT := 16#00000031;
END_VAR
CASE iState OF
0: (* idle *)
	IF Execute AND NOT bExecute_I THEN
		bExecute_I := Execute;

		(* use axis id to determine stDriveRef *)
		IF (Axis.NcToPlc.AxisId = nAxisId_I) AND (stDriveRef.nSlaveAddr <> 0)  AND (stDriveRef.sNetId <> '') THEN
			(* Axis ID unchanged, reference available *)
			iState := 20; (* use reference *)
		ELSE
			(* Axis ID changed *)
			iState := 10; (* get reference from NC *)
			MEMSET(ADR(stDriveRef), 0, SIZEOF(stDriveRef));
			MEMSET(ADR(readBuffer), 0, SIZEOF(readBuffer));

			fbAdsRead(
				NETID	:= NetId,
				PORT	:= AMSPORT_R0_NC,
				IDXGRP	:= NCIDXG_AXPARMS + Axis.NcToPlc.AxisId,
				IDXOFFS	:= NCIDXO_AXP_HWAMSADDR,
				LEN		:= SIZEOF(readBuffer) ,
				DESTADDR:= ADR(readBuffer),
				READ	:= FALSE,
				TMOUT	:= Timeout
			);
			fbAdsRead(READ := TRUE);

		END_IF

		nAxisId_I 	:= Axis.NcToPlc.AxisId;
		Busy		:= TRUE;
		Error		:= FALSE;
		AdsErrId	:= 0;
		SercosErrId	:= 0;
	END_IF

10: (* get reference from NC *)
	fbAdsRead(READ := FALSE);
	IF NOT fbAdsRead.BUSY THEN
		fbAdsRead(READ := FALSE);

		IF NOT fbAdsRead.ERR THEN
			MEMCPY(ADR(nIds), ADR(readBuffer), SIZEOF(nIds)); 										(* readBuffer[0..5] *)
			MEMCPY(ADR(stDriveRef.nSlaveAddr), ADR(readBuffer[6]), SIZEOF(stDriveRef.nSlaveAddr));  	(* readBuffer[6..7] *)
			MEMCPY(ADR(stDriveRef.nDriveNo), ADR(readBuffer[8]), SIZEOF(stDriveRef.nDriveNo));  		(* readBuffer[8..9] *)

			(* create string out of byte array *)
			stDriveRef.sNetId := F_CreateAmsNetId(nIds);
			iState	:= 20;
		ELSE
			Busy	:= FALSE;
			Error	:= TRUE;
			AdsErrId	:= UDINT_TO_UINT(fbAdsRead.ERRID);
			iState	:= 0;
			Attribute := 0;
			DcBusVoltage := 0;
		END_IF
	END_IF

20: (* read DC bus voltage *)
	fbEcSoEReadDcBusVolt(
		stDriveRef		:= stDriveRef,
		bExecute		:= FALSE,
		tTimeout		:= Timeout
	);
	fbEcSoEReadDcBusVolt(bExecute := TRUE);
	iState	:= 30;

30: (* wait for read DC bus voltage done *)
	fbEcSoEReadDcBusVolt(bExecute := FALSE);

	IF NOT fbEcSoEReadDcBusVolt.bBusy THEN
		fbEcSoEReadDcBusVolt(bExecute := FALSE);
		iState	:= 0;

		IF NOT fbEcSoEReadDcBusVolt.bError THEN
			Busy	:= FALSE;
			DcBusVoltage := fbEcSoEReadDcBusVolt.fDcBusVoltage;
			Attribute := fbEcSoEReadDcBusVolt.dwAttribute;
		ELSE
			Busy	:= FALSE;
			Error	:= TRUE;
			AdsErrId		:= fbEcSoEReadDcBusVolt.iAdsErrId;
			SercosErrId	:= fbEcSoEReadDcBusVolt.iSercosErrId;
			Attribute 	:= fbEcSoEReadDcBusVolt.dwAttribute;
			DcBusVoltage := 0;
		END_IF
	END_IF

END_CASE

bExecute_I := bExecute_I AND Execute;
END_FUNCTION_BLOCK

(* POU FB_SoEReadDiagMessage, ST *)
FUNCTION_BLOCK FB_SoEReadDiagMessage
VAR_INPUT
	NetId			: T_AmsNetId := '';	(* netID of PC with NC *)
	Execute			: BOOL;				(* Function block execution is triggered by a rising edge at this input.*)
	Timeout			: TIME := DEFAULT_ADS_TIMEOUT;(* States the time before the function is cancelled. *)
END_VAR
VAR_IN_OUT
	Axis			: AXIS_REF;	(* Axis reference *)
END_VAR
VAR_OUTPUT
	Busy			: BOOL;
	Error			: BOOL;
	AdsErrId		: UINT;
	SercosErrId		: UINT;
	DiagMessage		: ST_SoE_String;
	Attribute		: DWORD;
END_VAR
{library private}
VAR
	fbEcSoEReadDiag	: FB_SoEReadDiagMessage_ByDriveRef;
	iState			: INT;
	bExecute_I		: BOOL;
   	nAxisId_I      	: DWORD;
	fbAdsRead		: ADSREAD;
	readBuffer		: ARRAY[0..9] OF BYTE;
	nIds			: T_AmsNetIdArr; (* Ams net id as array of bytes *)
	stDriveRef		: ST_DriveRef; (* contains sNetID of EcMaster, nSlaveAddr of EcDrive, nDriveNo of EcDrive, either preset or read from NC *)
END_VAR
VAR CONSTANT
	NCIDXG_AXPARMS			: UDINT := 16#00004000;	(* Axis with ID: Parameter 			*)
	NCIDXO_AXP_HWAMSADDR	: UDINT := 16#00000031;
END_VAR
CASE iState OF
0: (* idle *)
	IF Execute AND NOT bExecute_I THEN
		bExecute_I := Execute;

		(* use axis id to determine stDriveRef *)
		IF (Axis.NcToPlc.AxisId = nAxisId_I) AND (stDriveRef.nSlaveAddr <> 0)  AND (stDriveRef.sNetId <> '') THEN
			(* Axis ID unchanged, reference available *)
			iState := 20; (* use reference *)
		ELSE
			(* Axis ID changed *)
			iState := 10; (* get reference from NC *)
			MEMSET(ADR(stDriveRef), 0, SIZEOF(stDriveRef));
			MEMSET(ADR(readBuffer), 0, SIZEOF(readBuffer));

			fbAdsRead(
				NETID	:= NetId,
				PORT	:= AMSPORT_R0_NC,
				IDXGRP	:= NCIDXG_AXPARMS + Axis.NcToPlc.AxisId,
				IDXOFFS	:= NCIDXO_AXP_HWAMSADDR,
				LEN		:= SIZEOF(readBuffer) ,
				DESTADDR:= ADR(readBuffer),
				READ	:= FALSE,
				TMOUT	:= Timeout
			);
			fbAdsRead(READ := TRUE);

		END_IF

		nAxisId_I 	:= Axis.NcToPlc.AxisId;
		Busy		:= TRUE;
		Error		:= FALSE;
		AdsErrId	:= 0;
		SercosErrId	:= 0;
	END_IF

10: (* get reference from NC *)
	fbAdsRead(READ := FALSE);
	IF NOT fbAdsRead.BUSY THEN
		fbAdsRead(READ := FALSE);

		IF NOT fbAdsRead.ERR THEN
			MEMCPY(ADR(nIds), ADR(readBuffer), SIZEOF(nIds)); 										(* readBuffer[0..5] *)
			MEMCPY(ADR(stDriveRef.nSlaveAddr), ADR(readBuffer[6]), SIZEOF(stDriveRef.nSlaveAddr));  	(* readBuffer[6..7] *)
			MEMCPY(ADR(stDriveRef.nDriveNo), ADR(readBuffer[8]), SIZEOF(stDriveRef.nDriveNo));  		(* readBuffer[8..9] *)

			(* create string out of byte array *)
			stDriveRef.sNetId := F_CreateAmsNetId(nIds);
			iState	:= 20;
		ELSE
			Busy	:= FALSE;
			Error	:= TRUE;
			AdsErrId:= UDINT_TO_UINT(fbAdsRead.ERRID);
			iState	:= 0;
			Attribute := 0;
			MEMSET(ADR(DiagMessage), 0, SIZEOF(DiagMessage));
		END_IF
	END_IF

20: (* read drive diag *)
	fbEcSoEReadDiag(
		stDriveRef		:= stDriveRef,
		bExecute		:= FALSE,
		tTimeout		:= Timeout
	);
	fbEcSoEReadDiag(bExecute := TRUE);
	iState	:= 30;

30: (* wait for read drive diag done *)
	fbEcSoEReadDiag(bExecute := FALSE);

	IF NOT fbEcSoEReadDiag.bBusy THEN
		fbEcSoEReadDiag(bExecute := FALSE);
		iState	:= 0;

		IF NOT fbEcSoEReadDiag.bError THEN
			Busy	:= FALSE;
			DiagMessage := fbEcSoEReadDiag.sDiagMessage;
			Attribute := fbEcSoEReadDiag.dwAttribute;
		ELSE
			Busy	:= FALSE;
			Error	:= TRUE;
			AdsErrId	:= fbEcSoEReadDiag.iAdsErrId;
			SercosErrId	:= fbEcSoEReadDiag.iSercosErrId;
			Attribute 	:= fbEcSoEReadDiag.dwAttribute;
			MEMSET(ADR(DiagMessage), 0, SIZEOF(DiagMessage));
		END_IF
	END_IF

END_CASE

bExecute_I := bExecute_I AND Execute;
END_FUNCTION_BLOCK

(* POU FB_SoEReadDiagNumber, ST *)
FUNCTION_BLOCK FB_SoEReadDiagNumber
VAR_INPUT
	NetId			: T_AmsNetId := '';	(* netID of PC with NC *)
	Execute			: BOOL;				(* Function block execution is triggered by a rising edge at this input.*)
	Timeout			: TIME := DEFAULT_ADS_TIMEOUT;(* States the time before the function is cancelled. *)
END_VAR
VAR_IN_OUT
	Axis			: AXIS_REF;	(* Axis reference *)
END_VAR
VAR_OUTPUT
	Busy			: BOOL;
	Error			: BOOL;
	AdsErrId		: UINT;
	SercosErrId		: UINT;
	DiagNumber		: UDINT;
	Attribute		: DWORD;
END_VAR
{library private}
VAR
	fbEcSoEReadDiag	: FB_SoEReadDiagNumber_ByDriveRef;
	iState			: INT;
	bExecute_I		: BOOL;
   	nAxisId_I      	: DWORD;
	fbAdsRead		: ADSREAD;
	readBuffer		: ARRAY[0..9] OF BYTE;
	nIds			: T_AmsNetIdArr; (* Ams net id as array of bytes *)
	stDriveRef		: ST_DriveRef; (* contains sNetID of EcMaster, nSlaveAddr of EcDrive, nDriveNo of EcDrive, either preset or read from NC *)
END_VAR
VAR CONSTANT
	NCIDXG_AXPARMS			: UDINT := 16#00004000;	(* Axis with ID: Parameter 			*)
	NCIDXO_AXP_HWAMSADDR	: UDINT := 16#00000031;
END_VAR
CASE iState OF
0: (* idle *)
	IF Execute AND NOT bExecute_I THEN
		bExecute_I := Execute;

		(* use axis id to determine stDriveRef *)
		IF (Axis.NcToPlc.AxisId = nAxisId_I) AND (stDriveRef.nSlaveAddr <> 0)  AND (stDriveRef.sNetId <> '') THEN
			(* Axis ID unchanged, reference available *)
			iState := 20; (* use reference *)
		ELSE
			(* Axis ID changed *)
			iState := 10; (* get reference from NC *)
			MEMSET(ADR(stDriveRef), 0, SIZEOF(stDriveRef));
			MEMSET(ADR(readBuffer), 0, SIZEOF(readBuffer));

			fbAdsRead(
				NETID	:= NetId,
				PORT	:= AMSPORT_R0_NC,
				IDXGRP	:= NCIDXG_AXPARMS + Axis.NcToPlc.AxisId,
				IDXOFFS	:= NCIDXO_AXP_HWAMSADDR,
				LEN		:= SIZEOF(readBuffer) ,
				DESTADDR:= ADR(readBuffer),
				READ	:= FALSE,
				TMOUT	:= Timeout
			);
			fbAdsRead(READ := TRUE);

		END_IF

		nAxisId_I 	:= Axis.NcToPlc.AxisId;
		Busy		:= TRUE;
		Error		:= FALSE;
		AdsErrId	:= 0;
		SercosErrId	:= 0;
	END_IF

10: (* get reference from NC *)
	fbAdsRead(READ := FALSE);
	IF NOT fbAdsRead.BUSY THEN
		fbAdsRead(READ := FALSE);

		IF NOT fbAdsRead.ERR THEN
			MEMCPY(ADR(nIds), ADR(readBuffer), SIZEOF(nIds)); 										(* readBuffer[0..5] *)
			MEMCPY(ADR(stDriveRef.nSlaveAddr), ADR(readBuffer[6]), SIZEOF(stDriveRef.nSlaveAddr));  	(* readBuffer[6..7] *)
			MEMCPY(ADR(stDriveRef.nDriveNo), ADR(readBuffer[8]), SIZEOF(stDriveRef.nDriveNo));  		(* readBuffer[8..9] *)

			(* create string out of byte array *)
			stDriveRef.sNetId := F_CreateAmsNetId(nIds);
			iState	:= 20;
		ELSE
			Busy	:= FALSE;
			Error	:= TRUE;
			AdsErrId:= UDINT_TO_UINT(fbAdsRead.ERRID);
			iState	:= 0;
			Attribute := 0;
			DiagNumber := 0;
		END_IF
	END_IF

20: (* read drive diag number *)
	fbEcSoEReadDiag(
		stDriveRef		:= stDriveRef,
		bExecute		:= FALSE,
		tTimeout		:= Timeout
	);
	fbEcSoEReadDiag(bExecute := TRUE);
	iState	:= 30;

30: (* wait for read drive diag number done *)
	fbEcSoEReadDiag(bExecute := FALSE);

	IF NOT fbEcSoEReadDiag.bBusy THEN
		fbEcSoEReadDiag(bExecute := FALSE);
		iState	:= 0;

		IF NOT fbEcSoEReadDiag.bError THEN
			Busy	:= FALSE;
			DiagNumber := fbEcSoEReadDiag.iDiagNumber;
			Attribute := fbEcSoEReadDiag.dwAttribute;
		ELSE
			Busy	:= FALSE;
			Error	:= TRUE;
			AdsErrId	:= fbEcSoEReadDiag.iAdsErrId;
			SercosErrId	:= fbEcSoEReadDiag.iSercosErrId;
			Attribute 	:= fbEcSoEReadDiag.dwAttribute;
			DiagNumber 	:= 0;
		END_IF
	END_IF

END_CASE

bExecute_I := bExecute_I AND Execute;
END_FUNCTION_BLOCK

(* POU FB_SoEReadDiagNumberList, ST *)
FUNCTION_BLOCK FB_SoEReadDiagNumberList
VAR_INPUT
	NetId			: T_AmsNetId := '';	(* netID of PC with NC *)
	Execute			: BOOL;				(* Function block execution is triggered by a rising edge at this input.*)
	Timeout			: TIME := DEFAULT_ADS_TIMEOUT;(* States the time before the function is cancelled. *)
	pDiagNumber		: POINTER TO ST_SoE_DiagNumList;
	Size			: UDINT;
END_VAR
VAR_IN_OUT
	Axis			: AXIS_REF;	(* Axis reference *)
END_VAR
VAR_OUTPUT
	Busy			: BOOL;
	Error			: BOOL;
	AdsErrId		: UINT;
	SercosErrId		: UINT;
	Attribute		: DWORD;
END_VAR
{library private}
VAR
	fbEcSoEReadDiag	: FB_SoEReadDiagNumberList_ByDriveRef;
	iState			: INT;
	bExecute_I		: BOOL;
   	nAxisId_I      	: DWORD;
	fbAdsRead		: ADSREAD;
	readBuffer		: ARRAY[0..9] OF BYTE;
	nIds			: T_AmsNetIdArr; (* Ams net id as array of bytes *)
	stDriveRef		: ST_DriveRef; (* contains sNetID of EcMaster, nSlaveAddr of EcDrive, nDriveNo of EcDrive, either preset or read from NC *)
END_VAR
VAR CONSTANT
	NCIDXG_AXPARMS			: UDINT := 16#00004000;	(* Axis with ID: Parameter 			*)
	NCIDXO_AXP_HWAMSADDR	: UDINT := 16#00000031;
END_VAR
CASE iState OF
0: (* idle *)
	IF Execute AND NOT bExecute_I THEN
		bExecute_I := Execute;

		(* use axis id to determine stDriveRef *)
		IF (Axis.NcToPlc.AxisId = nAxisId_I) AND (stDriveRef.nSlaveAddr <> 0)  AND (stDriveRef.sNetId <> '') THEN
			(* Axis ID unchanged, reference available *)
			iState := 20; (* use reference *)
		ELSE
			(* Axis ID changed *)
			iState := 10; (* get reference from NC *)
			MEMSET(ADR(stDriveRef), 0, SIZEOF(stDriveRef));
			MEMSET(ADR(readBuffer), 0, SIZEOF(readBuffer));

			fbAdsRead(
				NETID	:= NetId,
				PORT	:= AMSPORT_R0_NC,
				IDXGRP	:= NCIDXG_AXPARMS + Axis.NcToPlc.AxisId,
				IDXOFFS	:= NCIDXO_AXP_HWAMSADDR,
				LEN		:= SIZEOF(readBuffer) ,
				DESTADDR:= ADR(readBuffer),
				READ	:= FALSE,
				TMOUT	:= Timeout
			);
			fbAdsRead(READ := TRUE);

		END_IF

		nAxisId_I 	:= Axis.NcToPlc.AxisId;
		Busy		:= TRUE;
		Error		:= FALSE;
		AdsErrId	:= 0;
		SercosErrId	:= 0;
	END_IF

10: (* get reference from NC *)
	fbAdsRead(READ := FALSE);
	IF NOT fbAdsRead.BUSY THEN
		fbAdsRead(READ := FALSE);

		IF NOT fbAdsRead.ERR THEN
			MEMCPY(ADR(nIds), ADR(readBuffer), SIZEOF(nIds)); 										(* readBuffer[0..5] *)
			MEMCPY(ADR(stDriveRef.nSlaveAddr), ADR(readBuffer[6]), SIZEOF(stDriveRef.nSlaveAddr)); 	(* readBuffer[6..7] *)
			MEMCPY(ADR(stDriveRef.nDriveNo), ADR(readBuffer[8]), SIZEOF(stDriveRef.nDriveNo));  	(* readBuffer[8..9] *)

			(* create string out of byte array *)
			stDriveRef.sNetId := F_CreateAmsNetId(nIds);
			iState	:= 20;
		ELSE
			Busy	:= FALSE;
			Error	:= TRUE;
			AdsErrId	:= UDINT_TO_UINT(fbAdsRead.ERRID);
			iState	:= 0;
			Attribute := 0;
			IF (pDiagNumber <> 0) AND (Size <> 0) THEN
				MEMSET(pDiagNumber, 0, Size);
			END_IF
		END_IF
	END_IF

20: (* read drive diag *)
	fbEcSoEReadDiag(
		stDriveRef		:= stDriveRef,
		bExecute		:= FALSE,
		tTimeout		:= Timeout,
		piDiagNumber	:= pDiagNumber,
		iSize			:= Size
	);
	fbEcSoEReadDiag(bExecute := TRUE);
	iState	:= 30;

30: (* wait for read drive diag done *)
	fbEcSoEReadDiag(bExecute := FALSE);

	IF NOT fbEcSoEReadDiag.bBusy THEN
		fbEcSoEReadDiag(bExecute := FALSE);
		iState	:= 0;

		IF NOT fbEcSoEReadDiag.bError THEN
			Busy	:= FALSE;
			Attribute := fbEcSoEReadDiag.dwAttribute;
		ELSE
			Busy	:= FALSE;
			Error	:= TRUE;
			AdsErrId	:= fbEcSoEReadDiag.iAdsErrId;
			SercosErrId	:= fbEcSoEReadDiag.iSercosErrId;
			Attribute 	:= fbEcSoEReadDiag.dwAttribute;
			IF (pDiagNumber <> 0) AND (Size <> 0) THEN
				MEMSET(pDiagNumber, 0, Size);
			END_IF
		END_IF
	END_IF

END_CASE

bExecute_I := bExecute_I AND Execute;
END_FUNCTION_BLOCK

(* POU FB_SoEReadMotorTemperature, ST *)
FUNCTION_BLOCK FB_SoEReadMotorTemperature
VAR_INPUT
	NetId					: T_AmsNetId := '';	(* netID of PC with NC *)
	Execute					: BOOL;				(* Function block execution is triggered by a rising edge at this input.*)
	Timeout					: TIME := DEFAULT_ADS_TIMEOUT;(* States the time before the function is cancelled. *)
END_VAR
VAR_IN_OUT
	Axis					: AXIS_REF;	(* Axis reference *)
END_VAR
VAR_OUTPUT
	Busy					: BOOL;
	Error					: BOOL;
	AdsErrId				: UINT;
	SercosErrId				: UINT;
	MotorTemperature		: REAL;
	Attribute				: DWORD;
END_VAR
{library private}
VAR
	fbEcSoEReadMotorTemp	: FB_SoEReadMotorTemperature_ByDriveRef;
	iState					: INT;
	bExecute_I				: BOOL;
   	nAxisId_I      			: DWORD;
	fbAdsRead				: ADSREAD;
	readBuffer				: ARRAY[0..9] OF BYTE;
	nIds					: T_AmsNetIdArr; (* Ams net id as array of bytes *)
	stDriveRef				: ST_DriveRef; (* contains sNetID of EcMaster, nSlaveAddr of EcDrive, nDriveNo of EcDrive, either preset or read from NC *)
END_VAR
VAR CONSTANT
	NCIDXG_AXPARMS			: UDINT := 16#00004000;	(* Axis with ID: Parameter 			*)
	NCIDXO_AXP_HWAMSADDR	: UDINT := 16#00000031;
END_VAR
CASE iState OF
0: (* idle *)
	IF Execute AND NOT bExecute_I THEN
		bExecute_I := Execute;

		(* use axis id to determine stDriveRef *)
		IF (Axis.NcToPlc.AxisId = nAxisId_I) AND (stDriveRef.nSlaveAddr <> 0)  AND (stDriveRef.sNetId <> '') THEN
			(* Axis ID unchanged, reference available *)
			iState := 20; (* use reference *)
		ELSE
			(* Axis ID changed *)
			iState := 10; (* get reference from NC *)
			MEMSET(ADR(stDriveRef), 0, SIZEOF(stDriveRef));
			MEMSET(ADR(readBuffer), 0, SIZEOF(readBuffer));

			fbAdsRead(
				NETID	:= NetId,
				PORT	:= AMSPORT_R0_NC,
				IDXGRP	:= NCIDXG_AXPARMS + Axis.NcToPlc.AxisId,
				IDXOFFS	:= NCIDXO_AXP_HWAMSADDR,
				LEN		:= SIZEOF(readBuffer) ,
				DESTADDR:= ADR(readBuffer),
				READ	:= FALSE,
				TMOUT	:= Timeout
			);
			fbAdsRead(READ := TRUE);

		END_IF

		nAxisId_I 	:= Axis.NcToPlc.AxisId;
		Busy		:= TRUE;
		Error		:= FALSE;
		AdsErrId	:= 0;
		SercosErrId	:= 0;
	END_IF

10: (* get reference from NC *)
	fbAdsRead(READ := FALSE);
	IF NOT fbAdsRead.BUSY THEN
		fbAdsRead(READ := FALSE);

		IF NOT fbAdsRead.ERR THEN
			MEMCPY(ADR(nIds), ADR(readBuffer), SIZEOF(nIds)); 										(* readBuffer[0..5] *)
			MEMCPY(ADR(stDriveRef.nSlaveAddr), ADR(readBuffer[6]), SIZEOF(stDriveRef.nSlaveAddr));  	(* readBuffer[6..7] *)
			MEMCPY(ADR(stDriveRef.nDriveNo), ADR(readBuffer[8]), SIZEOF(stDriveRef.nDriveNo));  		(* readBuffer[8..9] *)

			(* create string out of byte array *)
			stDriveRef.sNetId := F_CreateAmsNetId(nIds);
			iState	:= 20;
		ELSE
			Busy	:= FALSE;
			Error	:= TRUE;
			AdsErrId	:= UDINT_TO_UINT(fbAdsRead.ERRID);
			iState	:= 0;
			Attribute := 0;
			MotorTemperature := 0;
		END_IF
	END_IF

20: (* read Motor Temperature *)
	fbEcSoEReadMotorTemp(
		stDriveRef		:= stDriveRef,
		bExecute		:= FALSE,
		tTimeout		:= Timeout
	);
	fbEcSoEReadMotorTemp(bExecute := TRUE);
	iState	:= 30;

30: (* wait for read Motor Temperature done *)
	fbEcSoEReadMotorTemp(bExecute := FALSE);

	IF NOT fbEcSoEReadMotorTemp.bBusy THEN
		fbEcSoEReadMotorTemp(bExecute := FALSE);
		iState	:= 0;

		IF NOT fbEcSoEReadMotorTemp.bError THEN
			Busy	:= FALSE;
			Attribute 	  := fbEcSoEReadMotorTemp.dwAttribute;
			MotorTemperature := fbEcSoEReadMotorTemp.fMotorTemperature;
		ELSE
			Busy	:= FALSE;
			Error	:= TRUE;
			AdsErrId		:= fbEcSoEReadMotorTemp.iAdsErrId;
			SercosErrId		:= fbEcSoEReadMotorTemp.iSercosErrId;
			Attribute 		:= fbEcSoEReadMotorTemp.dwAttribute;
			MotorTemperature := 0;
		END_IF
	END_IF

END_CASE

bExecute_I := bExecute_I AND Execute;
END_FUNCTION_BLOCK

(* POU FB_SoEReset, ST *)
FUNCTION_BLOCK FB_SoEReset
VAR_INPUT
	NetId			: T_AmsNetId := '';	(* netID of PC with NC *)
	Execute			: BOOL;				(* Function block execution is triggered by a rising edge at this input.*)
	Timeout			: TIME := T#10s;	(* States the time before the function is cancelled. (up to 10s) *)
END_VAR
VAR_IN_OUT
	Axis			: AXIS_REF;	(* Axis reference *)
END_VAR
VAR_OUTPUT
	Busy			: BOOL;
	Error			: BOOL;
	AdsErrId		: UINT;
	SercosErrId		: UINT;
END_VAR
{library private}
VAR
	fbEcSoEReset	: FB_SoEReset_ByDriveRef;
	iState			: INT;
	bExecute_I		: BOOL;
   	nAxisId_I      	: DWORD;
	fbAdsRead		: ADSREAD;
	readBuffer		: ARRAY[0..9] OF BYTE;
	nIds			: T_AmsNetIdArr; (* Ams net id as array of bytes *)
	stDriveRef		: ST_DriveRef; (* contains sNetID of EcMaster, nSlaveAddr of EcDrive, nDriveNo of EcDrive, either preset or read from NC *)
END_VAR
VAR CONSTANT
	NCIDXG_AXPARMS			: UDINT := 16#00004000;	(* Axis with ID: Parameter 			*)
	NCIDXO_AXP_HWAMSADDR	: UDINT := 16#00000031;
END_VAR
CASE iState OF
0: (* idle *)
	IF Execute AND NOT bExecute_I THEN
		bExecute_I := Execute;

		(* use axis id to determine stDriveRef *)
		IF (Axis.NcToPlc.AxisId = nAxisId_I) AND (stDriveRef.nSlaveAddr <> 0)  AND (stDriveRef.sNetId <> '') THEN
			(* Axis ID unchanged, reference available *)
			iState := 20; (* use reference *)
		ELSE
			(* Axis ID changed *)
			iState := 10; (* get reference from NC *)
			MEMSET(ADR(stDriveRef), 0, SIZEOF(stDriveRef));
			MEMSET(ADR(readBuffer), 0, SIZEOF(readBuffer));

			fbAdsRead(
				NETID	:= NetId,
				PORT	:= AMSPORT_R0_NC,
				IDXGRP	:= NCIDXG_AXPARMS + Axis.NcToPlc.AxisId,
				IDXOFFS	:= NCIDXO_AXP_HWAMSADDR,
				LEN		:= SIZEOF(readBuffer) ,
				DESTADDR:= ADR(readBuffer),
				READ	:= FALSE,
				TMOUT	:= Timeout
			);
			fbAdsRead(READ := TRUE);

		END_IF

		nAxisId_I 	:= Axis.NcToPlc.AxisId;
		Busy		:= TRUE;
		Error		:= FALSE;
		AdsErrId	:= 0;
		SercosErrId	:= 0;
	END_IF

10: (* get reference from NC *)
	fbAdsRead(READ := FALSE);
	IF NOT fbAdsRead.BUSY THEN
		fbAdsRead(READ := FALSE);

		IF NOT fbAdsRead.ERR THEN
			MEMCPY(ADR(nIds), ADR(readBuffer), SIZEOF(nIds)); 										(* readBuffer[0..5] *)
			MEMCPY(ADR(stDriveRef.nSlaveAddr), ADR(readBuffer[6]), SIZEOF(stDriveRef.nSlaveAddr));  (* readBuffer[6..7] *)
			MEMCPY(ADR(stDriveRef.nDriveNo), ADR(readBuffer[8]), SIZEOF(stDriveRef.nDriveNo));  	(* readBuffer[8..9] *)

			(* create string out of byte array *)
			stDriveRef.sNetId := F_CreateAmsNetId(nIds);
			iState	:= 20;
		ELSE
			Busy	:= FALSE;
			Error	:= TRUE;
			AdsErrId	:= UDINT_TO_UINT(fbAdsRead.ERRID);
			iState	:= 0;
		END_IF
	END_IF

20: (* reset drive *)
	fbEcSoEReset(
		stDriveRef	:= stDriveRef,
		bExecute	:= FALSE,
		tTimeout	:= Timeout
	);
	fbEcSoEReset(bExecute := TRUE);
	iState	:= 30;

30: (* wait for drive reset done *)
	fbEcSoEReset(bExecute := FALSE);

	IF NOT fbEcSoEReset.bBusy THEN
		fbEcSoEReset(bExecute := FALSE);

		IF NOT fbEcSoEReset.bError THEN
			iState		:= 0;
			Busy		:= FALSE;
			Error		:= FALSE;
		ELSE
			iState		:= 0;
			Busy		:= FALSE;
			Error		:= TRUE;
			AdsErrId	:= fbEcSoEReset.iAdsErrId;
			SercosErrId	:= fbEcSoEReset.iSercosErrId;
		END_IF
	END_IF

END_CASE

bExecute_I := bExecute_I AND Execute;
END_FUNCTION_BLOCK

(* POU FB_SoEWrite, ST *)
FUNCTION_BLOCK FB_SoEWrite
VAR_INPUT
	NetId			: T_AmsNetId := '';	(* netID of PC with NC *)
	Idn				: WORD;		(* SoE IDN: e.g. "S_0_IDN + 1" for S-0-0001 or "P_0_IDN + 23" for P-0-0023*)
	Element			: BYTE;		(* SoE element.*)
	pSrcBuf			: DWORD;	(* Contains the address of the buffer containing the data to be send. *)
	BufLen			: UDINT;	(* Contains the max. number of bytes to be received. *)
	Execute			: BOOL;				(* Function block execution is triggered by a rising edge at this input.*)
	Timeout			: TIME := DEFAULT_ADS_TIMEOUT;(* States the time before the function is cancelled. *)
	Password		: ST_SoE_String;
END_VAR
VAR_IN_OUT
	Axis			: AXIS_REF;	(* Axis reference *)
END_VAR
VAR_OUTPUT
	Busy			: BOOL;
	Error			: BOOL;
	AdsErrId		: UINT;
	SercosErrId		: UINT;
END_VAR
{library private}
VAR
	fbEcSoEWriteEx	: FB_SoEWrite_ByDriveRef;
	iState			: INT;
	bExecute_I		: BOOL;
   	nAxisId_I      	: DWORD;
	fbAdsRead		: ADSREAD;
	readBuffer		: ARRAY[0..9] OF BYTE;
	nIds			: T_AmsNetIdArr; (* Ams net id as array of bytes *)
	stDriveRef		: ST_DriveRef; (* contains sNetID of EcMaster, nSlaveAddr of EcDrive, nDriveNo of EcDrive, either preset or read from NC *)
END_VAR
VAR CONSTANT
	NCIDXG_AXPARMS			: UDINT := 16#00004000;	(* Axis with ID: Parameter 			*)
	NCIDXO_AXP_HWAMSADDR	: UDINT := 16#00000031;
END_VAR
CASE iState OF
0: (* idle *)
	IF Execute AND NOT bExecute_I THEN
		bExecute_I := Execute;

		(* use axis id to determine stDriveRef *)
		IF (Axis.NcToPlc.AxisId = nAxisId_I) AND (stDriveRef.nSlaveAddr <> 0)  AND (stDriveRef.sNetId <> '') THEN
			(* Axis ID unchanged, reference available *)
			iState := 20; (* use reference *)
		ELSE
			(* Axis ID changed *)
			iState := 10; (* get reference from NC *)
			MEMSET(ADR(stDriveRef), 0, SIZEOF(stDriveRef));
			MEMSET(ADR(readBuffer), 0, SIZEOF(readBuffer));

			fbAdsRead(
				NETID	:= NetId,
				PORT	:= AMSPORT_R0_NC,
				IDXGRP	:= NCIDXG_AXPARMS + Axis.NcToPlc.AxisId,
				IDXOFFS	:= NCIDXO_AXP_HWAMSADDR,
				LEN		:= SIZEOF(readBuffer) ,
				DESTADDR:= ADR(readBuffer),
				READ	:= FALSE,
				TMOUT	:= Timeout
			);
			fbAdsRead(READ := TRUE);

		END_IF

		nAxisId_I 	:= Axis.NcToPlc.AxisId;
		Busy		:= TRUE;
		Error		:= FALSE;
		AdsErrId	:= 0;
		SercosErrId	:= 0;
	END_IF

10: (* get reference from NC *)
	fbAdsRead(READ := FALSE);
	IF NOT fbAdsRead.BUSY THEN
		fbAdsRead(READ := FALSE);

		IF NOT fbAdsRead.ERR THEN
			MEMCPY(ADR(nIds), ADR(readBuffer), SIZEOF(nIds)); 										(* readBuffer[0..5] *)
			MEMCPY(ADR(stDriveRef.nSlaveAddr), ADR(readBuffer[6]), SIZEOF(stDriveRef.nSlaveAddr));  	(* readBuffer[6..7] *)
			MEMCPY(ADR(stDriveRef.nDriveNo), ADR(readBuffer[8]), SIZEOF(stDriveRef.nDriveNo));  		(* readBuffer[8..9] *)

			(* create string out of byte array *)
			stDriveRef.sNetId := F_CreateAmsNetId(nIds);
			iState	:= 20;
		ELSE
			Busy	:= FALSE;
			Error	:= TRUE;
			AdsErrId	:= UDINT_TO_UINT(fbAdsRead.ERRID);
			iState	:= 0;
		END_IF
	END_IF

20: (* write SoE data *)
	fbEcSoEWriteEx(
		stDriveRef		:= stDriveRef,
		nIdn			:= Idn,
		nElement		:= Element,
		pSrcBuf			:= pSrcBuf,
		cbBufLen		:= BufLen,
		bExecute		:= FALSE,
		tTimeout		:= Timeout
	);
	fbEcSoEWriteEx(bExecute := TRUE);
	iState	:= 30;

30: (* wait for write SoE data done *)
	fbEcSoEWriteEx(bExecute := FALSE);

	IF NOT fbEcSoEWriteEx.bBusy THEN
		fbEcSoEWriteEx(bExecute := FALSE);
		iState	:= 0;

		IF NOT fbEcSoEWriteEx.bError THEN
			Busy	:= FALSE;
		ELSE
			Busy	:= FALSE;
			Error	:= TRUE;
			AdsErrId	:= fbEcSoEWriteEx.iAdsErrId;
			SercosErrId	:= fbEcSoEWriteEx.iSercosErrId;
		END_IF
	END_IF

END_CASE

bExecute_I := bExecute_I AND Execute;
END_FUNCTION_BLOCK

(* POU FB_SoEWriteCommandControl, ST *)
FUNCTION_BLOCK FB_SoEWriteCommandControl
VAR_INPUT
	NetId			: T_AmsNetId := '';	(* netID of PC with NC *)
	Idn				: WORD;		(* SoE IDN: e.g. "S_0_IDN + 1" for S-0-0001 or "P_0_IDN + 23" for P-0-0023*)
	CmdControl		: E_SoE_CmdControl;	(* eSoE_CmdControl_Cancel, eSoE_CmdControl_Set, eSoE_CmdControl_SetAndEnable*)
	Execute			: BOOL;				(* Function block execution is triggered by a rising edge at this input.*)
	Timeout			: TIME := DEFAULT_ADS_TIMEOUT;(* States the time before the function is cancelled. *)
END_VAR
VAR_IN_OUT
	Axis			: AXIS_REF;	(* Axis reference *)
END_VAR
VAR_OUTPUT
	Busy			: BOOL;
	Error			: BOOL;
	AdsErrId		: UINT;
	SercosErrId		: UINT;
END_VAR
{library private}
VAR
	fbEcSoECommand	: FB_SoEWriteCommandControl_ByDriveRef;
	iState			: INT;
	bExecute_I		: BOOL;
   	nAxisId_I      	: DWORD;
	fbAdsRead		: ADSREAD;
	readBuffer		: ARRAY[0..9] OF BYTE;
	nIds			: T_AmsNetIdArr; (* Ams net id as array of bytes *)
	stDriveRef		: ST_DriveRef; (* contains sNetID of EcMaster, nSlaveAddr of EcDrive, nDriveNo of EcDrive, either preset or read from NC *)
END_VAR
VAR CONSTANT
	NCIDXG_AXPARMS			: UDINT := 16#00004000;	(* Axis with ID: Parameter 			*)
	NCIDXO_AXP_HWAMSADDR	: UDINT := 16#00000031;
END_VAR
CASE iState OF
0: (* idle *)
	IF Execute AND NOT bExecute_I THEN
		bExecute_I := Execute;

		(* use axis id to determine stDriveRef *)
		IF (Axis.NcToPlc.AxisId = nAxisId_I) AND (stDriveRef.nSlaveAddr <> 0)  AND (stDriveRef.sNetId <> '') THEN
			(* Axis ID unchanged, reference available *)
			iState := 20; (* use reference *)
		ELSE
			(* Axis ID changed *)
			iState := 10; (* get reference from NC *)
			MEMSET(ADR(stDriveRef), 0, SIZEOF(stDriveRef));
			MEMSET(ADR(readBuffer), 0, SIZEOF(readBuffer));

			fbAdsRead(
				NETID	:= NetId,
				PORT	:= AMSPORT_R0_NC,
				IDXGRP	:= NCIDXG_AXPARMS + Axis.NcToPlc.AxisId,
				IDXOFFS	:= NCIDXO_AXP_HWAMSADDR,
				LEN		:= SIZEOF(readBuffer) ,
				DESTADDR:= ADR(readBuffer),
				READ	:= FALSE,
				TMOUT	:= Timeout
			);
			fbAdsRead(READ := TRUE);

		END_IF

		nAxisId_I 	:= Axis.NcToPlc.AxisId;
		Busy		:= TRUE;
		Error		:= FALSE;
		AdsErrId	:= 0;
		SercosErrId	:= 0;
	END_IF

10: (* get reference from NC *)
	fbAdsRead(READ := FALSE);
	IF NOT fbAdsRead.BUSY THEN
		fbAdsRead(READ := FALSE);

		IF NOT fbAdsRead.ERR THEN
			MEMCPY(ADR(nIds), ADR(readBuffer), SIZEOF(nIds)); 										(* readBuffer[0..5] *)
			MEMCPY(ADR(stDriveRef.nSlaveAddr), ADR(readBuffer[6]), SIZEOF(stDriveRef.nSlaveAddr));  	(* readBuffer[6..7] *)
			MEMCPY(ADR(stDriveRef.nDriveNo), ADR(readBuffer[8]), SIZEOF(stDriveRef.nDriveNo));  		(* readBuffer[8..9] *)

			(* create string out of byte array *)
			stDriveRef.sNetId := F_CreateAmsNetId(nIds);
			iState	:= 20;
		ELSE
			Busy	:= FALSE;
			Error	:= TRUE;
			AdsErrId:= UDINT_TO_UINT(fbAdsRead.ERRID);
			iState	:= 0;
		END_IF
	END_IF

20: (* write SoE command *)
	fbEcSoECommand(
		stDriveRef		:= stDriveRef,
		nIdn			:= Idn,
		eCmdControl		:= CmdControl,
		bExecute		:= FALSE,
		tTimeout		:= Timeout
	);
	fbEcSoECommand(bExecute := TRUE);
	iState	:= 30;

30: (* wait for write SoE command done *)
	fbEcSoECommand(bExecute := FALSE);

	IF NOT fbEcSoECommand.bBusy THEN
		fbEcSoECommand(bExecute := FALSE);
		iState	:= 0;

		IF NOT fbEcSoECommand.bError THEN
			Busy	:= FALSE;
		ELSE
			Busy	:= FALSE;
			Error	:= TRUE;
			AdsErrId	:= fbEcSoECommand.iAdsErrId;
			SercosErrId	:= fbEcSoECommand.iSercosErrId;
		END_IF
	END_IF

END_CASE

bExecute_I := bExecute_I AND Execute;
END_FUNCTION_BLOCK

(* POU FB_SoEWritePassword, ST *)
FUNCTION_BLOCK FB_SoEWritePassword
VAR_INPUT
	NetId			: T_AmsNetId := '';	(* netID of PC with NC *)
	Execute			: BOOL;				(* Function block execution is triggered by a rising edge at this input.*)
	Timeout			: TIME := DEFAULT_ADS_TIMEOUT;(* States the time before the function is cancelled. *)
	Password		: ST_SoE_String;
END_VAR
VAR_IN_OUT
	Axis			: AXIS_REF;	(* Axis reference *)
END_VAR
VAR_OUTPUT
	Busy			: BOOL;
	Error			: BOOL;
	AdsErrId		: UINT;
	SercosErrId		: UINT;
END_VAR
{library private}
VAR
	fbEcSoEWritePW	: FB_SoEWritePassword_ByDriveRef;
	iState			: INT;
	bExecute_I		: BOOL;
   	nAxisId_I      	: DWORD;
	fbAdsRead		: ADSREAD;
	readBuffer		: ARRAY[0..9] OF BYTE;
	nIds			: T_AmsNetIdArr; (* Ams net id as array of bytes *)
	stDriveRef		: ST_DriveRef; (* contains sNetID of EcMaster, nSlaveAddr of EcDrive, nDriveNo of EcDrive, either preset or read from NC *)
END_VAR
VAR CONSTANT
	NCIDXG_AXPARMS			: UDINT := 16#00004000;	(* Axis with ID: Parameter 			*)
	NCIDXO_AXP_HWAMSADDR	: UDINT := 16#00000031;
END_VAR
CASE iState OF
0: (* idle *)
	IF Execute AND NOT bExecute_I THEN
		bExecute_I := Execute;

		(* use axis id to determine stDriveRef *)
		IF (Axis.NcToPlc.AxisId = nAxisId_I) AND (stDriveRef.nSlaveAddr <> 0)  AND (stDriveRef.sNetId <> '') THEN
			(* Axis ID unchanged, reference available *)
			iState := 20; (* use reference *)
		ELSE
			(* Axis ID changed *)
			iState := 10; (* get reference from NC *)
			MEMSET(ADR(stDriveRef), 0, SIZEOF(stDriveRef));
			MEMSET(ADR(readBuffer), 0, SIZEOF(readBuffer));

			fbAdsRead(
				NETID	:= NetId,
				PORT	:= AMSPORT_R0_NC,
				IDXGRP	:= NCIDXG_AXPARMS + Axis.NcToPlc.AxisId,
				IDXOFFS	:= NCIDXO_AXP_HWAMSADDR,
				LEN		:= SIZEOF(readBuffer) ,
				DESTADDR:= ADR(readBuffer),
				READ	:= FALSE,
				TMOUT	:= Timeout
			);
			fbAdsRead(READ := TRUE);

		END_IF

		nAxisId_I 	:= Axis.NcToPlc.AxisId;
		Busy		:= TRUE;
		Error		:= FALSE;
		AdsErrId	:= 0;
		SercosErrId	:= 0;
	END_IF

10: (* get reference from NC *)
	fbAdsRead(READ := FALSE);
	IF NOT fbAdsRead.BUSY THEN
		fbAdsRead(READ := FALSE);

		IF NOT fbAdsRead.ERR THEN
			MEMCPY(ADR(nIds), ADR(readBuffer), SIZEOF(nIds)); 										(* readBuffer[0..5] *)
			MEMCPY(ADR(stDriveRef.nSlaveAddr), ADR(readBuffer[6]), SIZEOF(stDriveRef.nSlaveAddr));  	(* readBuffer[6..7] *)
			MEMCPY(ADR(stDriveRef.nDriveNo), ADR(readBuffer[8]), SIZEOF(stDriveRef.nDriveNo));  		(* readBuffer[8..9] *)

			(* create string out of byte array *)
			stDriveRef.sNetId := F_CreateAmsNetId(nIds);
			iState	:= 20;
		ELSE
			Busy	:= FALSE;
			Error	:= TRUE;
			AdsErrId:= UDINT_TO_UINT(fbAdsRead.ERRID);
			iState	:= 0;
		END_IF
	END_IF

20: (* write drive password *)
	fbEcSoEWritePW(
		stDriveRef		:= stDriveRef,
		bExecute		:= FALSE,
		tTimeout		:= Timeout,
		sPassword		:= Password
	);
	fbEcSoEWritePW(bExecute := TRUE);
	iState	:= 30;

30: (* wait for write drive password done *)
	fbEcSoEWritePW(bExecute := FALSE);

	IF NOT fbEcSoEWritePW.bBusy THEN
		fbEcSoEWritePW(bExecute := FALSE);
		iState	:= 0;

		IF NOT fbEcSoEWritePW.bError THEN
			Busy	:= FALSE;
		ELSE
			Busy	:= FALSE;
			Error	:= TRUE;
			AdsErrId	:= fbEcSoEWritePW.iAdsErrId;
			SercosErrId	:= fbEcSoEWritePW.iSercosErrId;
		END_IF
	END_IF

END_CASE

bExecute_I := bExecute_I AND Execute;
END_FUNCTION_BLOCK
